C07319=1167.736,-18.694,-45.324,179.712,5.920,149.143
C07320=1167.731,-18.445,-45.336,179.714,5.921,149.143
C07321=1167.726,-18.196,-45.349,179.717,5.921,149.142
C07322=1167.720,-17.945,-45.362,179.719,5.922,149.141
C07323=1167.715,-17.695,-45.374,179.722,5.922,149.141
C07324=1167.710,-17.446,-45.387,179.724,5.923,149.140
C07325=1167.705,-17.197,-45.399,179.726,5.923,149.140
C07326=1167.700,-16.947,-45.412,179.728,5.923,149.139
C07327=1167.694,-16.697,-45.426,179.731,5.924,149.138
C07328=1167.689,-16.448,-45.438,179.733,5.925,149.138
C07329=1167.684,-16.198,-45.451,179.736,5.925,149.137
C07330=1167.680,-15.948,-45.464,179.738,5.926,149.137
C07331=1167.674,-15.698,-45.476,179.741,5.926,149.136
C07332=1167.668,-15.449,-45.489,179.743,5.927,149.135
C07333=1167.663,-15.200,-45.501,179.746,5.928,149.135
C07334=1167.659,-14.950,-45.514,179.748,5.928,149.134
C07335=1167.654,-14.700,-45.527,179.751,5.928,149.133
C07336=1167.648,-14.451,-45.540,179.753,5.929,149.133
C07337=1167.643,-14.201,-45.553,179.756,5.930,149.132
C07338=1167.638,-13.951,-45.566,179.758,5.930,149.132
C07339=1167.633,-13.702,-45.578,179.761,5.931,149.131
C07340=1167.627,-13.452,-45.592,179.763,5.931,149.130
C07341=1167.623,-13.202,-45.604,179.765,5.932,149.130
C07342=1167.617,-12.953,-45.617,179.768,5.933,149.129
C07343=1167.612,-12.703,-45.630,179.770,5.933,149.129
C07344=1167.607,-12.453,-45.643,179.773,5.934,149.128
C07345=1167.602,-12.204,-45.656,179.776,5.934,149.127
C07346=1167.596,-11.954,-45.669,179.778,5.935,149.127
C07347=1167.591,-11.704,-45.682,179.780,5.936,149.126
C07348=1167.587,-11.456,-45.695,179.783,5.936,149.126
C07349=1167.582,-11.206,-45.708,179.785,5.937,149.125
C07350=1167.576,-10.956,-45.722,179.788,5.937,149.124
C07351=1167.571,-10.707,-45.734,179.790,5.938,149.124
C07352=1167.566,-10.457,-45.747,179.793,5.939,149.123
C07353=1167.561,-10.207,-45.760,179.795,5.939,149.123
C07354=1167.556,-9.958,-45.773,179.798,5.940,149.122
C07355=1167.550,-9.707,-45.786,179.800,5.940,149.121
C07356=1167.545,-9.458,-45.799,179.802,5.941,149.121
C07357=1167.540,-9.209,-45.812,179.805,5.942,149.120
C07358=1167.535,-8.959,-45.826,179.807,5.942,149.120
C07359=1167.530,-8.710,-45.839,179.810,5.943,149.119
C07360=1167.525,-8.460,-45.851,179.813,5.943,149.118
C07361=1167.520,-8.210,-45.865,179.815,5.944,149.118
C07362=1167.515,-7.961,-45.877,179.817,5.945,149.117
C07363=1167.510,-7.711,-45.892,179.820,5.945,149.117
C07364=1167.504,-7.462,-45.904,179.822,5.946,149.116
C07365=1167.499,-7.212,-45.917,179.825,5.946,149.115
C07366=1167.494,-6.962,-45.930,179.827,5.947,149.115
C07367=1167.489,-6.713,-45.943,179.830,5.948,149.114
C07368=1167.484,-6.463,-45.957,179.832,5.948,149.114
C07369=1167.479,-6.214,-45.970,179.834,5.949,149.113
C07370=1167.474,-5.963,-45.983,179.837,5.949,149.112
C07371=1167.469,-5.714,-45.996,179.839,5.950,149.112
C07372=1167.463,-5.465,-46.010,179.842,5.951,149.111
C07373=1167.458,-5.215,-46.023,179.844,5.951,149.111
C07374=1167.453,-4.966,-46.035,179.847,5.952,149.110
C07375=1167.448,-4.716,-46.050,179.849,5.952,149.109
C07376=1167.443,-4.467,-46.062,179.852,5.953,149.109
C07377=1167.438,-4.216,-46.076,179.854,5.954,149.108
C07378=1167.433,-3.967,-46.088,179.856,5.954,149.108
C07379=1167.427,-3.718,-46.102,179.859,5.955,149.107
C07380=1167.423,-3.468,-46.115,179.862,5.955,149.106
C07381=1167.417,-3.218,-46.129,179.864,5.956,149.106
C07382=1167.413,-2.969,-46.142,179.867,5.957,149.105
C07383=1167.407,-2.719,-46.155,179.869,5.957,149.105
C07384=1167.402,-2.470,-46.170,179.871,5.958,149.104
C07385=1167.397,-2.220,-46.182,179.874,5.960,149.104
C07386=1167.391,-1.970,-46.196,179.877,5.960,149.103
C07387=1167.387,-1.721,-46.209,179.880,5.960,149.102
C07388=1167.381,-1.471,-46.223,179.882,5.961,149.102
C07389=1167.376,-1.222,-46.235,179.884,5.962,149.101
C07390=1167.371,-0.972,-46.250,179.887,5.963,149.101
C07391=1167.366,-0.723,-46.262,179.889,5.963,149.100
C07392=1167.361,-0.473,-46.276,179.892,5.963,149.099
C07393=1167.355,-0.223,-46.290,179.894,5.964,149.099
C07394=1167.351,0.026,-46.303,179.897,5.965,149.098
C07395=1167.345,0.276,-46.317,179.899,5.966,149.098
C07396=1167.341,0.525,-46.330,179.901,5.966,149.097
C07397=1167.335,0.775,-46.343,179.904,5.967,149.096
C07398=1167.330,1.024,-46.358,179.906,5.967,149.096
C07399=1167.325,1.274,-46.370,179.909,5.968,149.095
C07400=1167.320,1.523,-46.385,179.911,5.969,149.095
C07401=1167.314,1.794,-46.399,179.914,5.970,149.094
C07402=1167.309,2.062,-46.413,179.917,5.970,149.093
C07403=1167.304,2.331,-46.428,179.920,5.971,149.093
C07404=1167.298,2.601,-46.443,179.922,5.971,149.092
C07405=1167.292,2.850,-46.456,179.925,5.972,149.091
C07406=1167.288,3.100,-46.470,179.927,5.973,149.091
C07407=1167.283,3.350,-46.483,179.929,5.973,149.090
C07408=1167.277,3.599,-46.497,179.933,5.975,149.090
C07409=1167.273,3.849,-46.510,179.935,5.975,149.089
C07410=1167.267,4.098,-46.524,179.937,5.976,149.088
C07411=1167.262,4.348,-46.538,179.940,5.976,149.088
C07412=1167.257,4.597,-46.552,179.942,5.977,149.087
C07413=1167.252,4.847,-46.565,179.945,5.978,149.087
C07414=1167.247,5.097,-46.579,179.948,5.978,149.086
C07415=1167.241,5.346,-46.593,179.950,5.979,149.085
C07416=1167.237,5.596,-46.606,179.952,5.979,149.085
C07417=1167.232,5.846,-46.620,179.955,5.980,149.084
C07418=1167.226,6.095,-46.634,179.957,5.981,149.084
C07419=1167.221,6.345,-46.648,179.960,5.981,149.083
C07420=1167.216,6.594,-46.661,179.963,5.983,149.082
C07421=1167.211,6.844,-46.675,179.965,5.983,149.082
C07422=1167.206,7.093,-46.689,179.967,5.984,149.081
C07423=1167.201,7.343,-46.703,179.970,5.985,149.081
C07424=1167.196,7.592,-46.716,179.972,5.985,149.080
C07425=1167.191,7.842,-46.730,179.975,5.986,149.079
C07426=1167.186,8.091,-46.744,179.978,5.986,149.079
C07427=1167.181,8.341,-46.758,179.980,5.987,149.078
C07428=1167.176,8.590,-46.771,179.982,5.988,149.078
C07429=1167.171,8.840,-46.786,179.985,5.988,149.077
C07430=1167.166,9.090,-46.800,179.988,5.990,149.076
C07431=1167.160,9.339,-46.813,179.990,5.990,149.076
C07432=1167.155,9.589,-46.827,179.993,5.991,149.075
C07433=1167.150,9.839,-46.842,179.995,5.992,149.075
C07434=1167.145,10.087,-46.855,179.997,5.992,149.074
C07435=1167.140,10.338,-46.868,-180.000,5.993,149.073
C07436=1167.135,10.587,-46.883,-179.997,5.993,149.073
C07437=1167.130,10.836,-46.897,-179.995,5.994,149.072
C07438=1167.125,11.086,-46.911,-179.992,5.995,149.072
C07439=1167.120,11.336,-46.925,-179.990,5.996,149.071
C07440=1167.115,11.585,-46.939,-179.987,5.997,149.071
C07441=1167.110,11.835,-46.952,-179.985,5.998,149.070
C07442=1167.105,12.085,-46.966,-179.982,5.998,149.069
C07443=1167.100,12.334,-46.981,-179.980,5.998,149.069
C07444=1167.094,12.583,-46.995,-179.977,5.999,149.068
C07445=1167.089,12.833,-47.009,-179.975,6.000,149.068
C07446=1167.084,13.083,-47.023,-179.973,6.001,149.067
C07447=1167.079,13.332,-47.037,-179.969,6.002,149.066
C07448=1167.074,13.581,-47.051,-179.967,6.002,149.066
C07449=1167.068,13.832,-47.065,-179.965,6.003,149.065
C07450=1167.064,14.081,-47.079,-179.962,6.004,149.065
C07451=1167.059,14.331,-47.093,-179.960,6.004,149.064
C07452=1167.054,14.580,-47.107,-179.957,6.005,149.063
C07453=1167.049,14.830,-47.121,-179.955,6.006,149.063
C07454=1167.044,15.079,-47.135,-179.952,6.006,149.062
C07455=1167.039,15.329,-47.150,-179.949,6.008,149.062
C07456=1167.033,15.578,-47.163,-179.947,6.008,149.061
C07457=1167.028,15.828,-47.178,-179.944,6.009,149.060
C07458=1167.023,16.077,-47.192,-179.942,6.010,149.060
C07459=1167.018,16.327,-47.206,-179.939,6.010,149.059
C07460=1167.013,16.576,-47.220,-179.937,6.011,149.059
C07461=1167.008,16.826,-47.234,-179.935,6.011,149.058
C07462=1167.003,17.076,-47.249,-179.931,6.013,149.058
C07463=1166.998,17.325,-47.263,-179.929,6.014,149.057
C07464=1166.993,17.575,-47.277,-179.927,6.014,149.056
C07465=1166.987,17.824,-47.291,-179.924,6.015,149.056
C07466=1166.982,18.074,-47.306,-179.922,6.015,149.055
C07467=1166.978,18.323,-47.320,-179.919,6.016,149.055
C07468=1166.973,18.573,-47.335,-179.916,6.017,149.054
C07469=1166.968,18.822,-47.349,-179.914,6.018,149.053
C07470=1166.962,19.071,-47.363,-179.911,6.019,149.053
C07471=1166.957,19.321,-47.377,-179.909,6.019,149.052
C07472=1166.952,19.571,-47.392,-179.907,6.020,149.052
C07473=1166.948,19.820,-47.406,-179.904,6.021,149.051
C07474=1166.942,20.070,-47.421,-179.901,6.022,149.050
C07475=1166.937,20.320,-47.435,-179.899,6.023,149.050
C07476=1166.931,20.569,-47.449,-179.896,6.023,149.049
C07477=1166.927,20.818,-47.464,-179.894,6.024,149.049
C07478=1166.922,21.068,-47.478,-179.891,6.024,149.048
C07479=1166.917,21.318,-47.492,-179.889,6.025,149.048
C07480=1166.912,21.567,-47.507,-179.886,6.027,149.047
C07481=1166.907,21.817,-47.521,-179.883,6.027,149.046
C07482=1166.902,22.066,-47.536,-179.881,6.028,149.046
C07483=1166.897,22.315,-47.550,-179.878,6.028,149.045
C07484=1166.891,22.565,-47.565,-179.876,6.029,149.045
C07485=1166.886,22.815,-47.579,-179.873,6.031,149.044
C07486=1166.881,23.065,-47.593,-179.871,6.031,149.044
C07487=1166.876,23.314,-47.608,-179.868,6.032,149.043
C07488=1166.871,23.563,-47.623,-179.865,6.032,149.042
C07489=1166.866,23.813,-47.637,-179.863,6.033,149.042
C07490=1166.861,24.062,-47.652,-179.861,6.034,149.041
C07491=1166.856,24.312,-47.667,-179.858,6.035,149.041
C07492=1166.851,24.561,-47.681,-179.855,6.036,149.040
C07493=1166.846,24.811,-47.695,-179.853,6.037,149.040
C07494=1166.841,25.060,-47.710,-179.850,6.037,149.039
C07495=1166.836,25.310,-47.724,-179.848,6.038,149.038
C07496=1166.830,25.560,-47.739,-179.845,6.039,149.038
C07497=1166.826,25.809,-47.754,-179.842,6.040,149.037
C07498=1166.821,26.059,-47.768,-179.840,6.041,149.037
C07499=1166.816,26.308,-47.783,-179.838,6.041,149.036
C07500=1166.810,26.558,-47.798,-179.835,6.043,149.036
C07501=1166.805,26.807,-47.812,-179.832,6.043,149.035
C07502=1166.800,27.057,-47.827,-179.830,6.044,149.034
C07503=1166.796,27.306,-47.842,-179.827,6.044,149.034
C07504=1166.790,27.556,-47.857,-179.825,6.045,149.033
C07505=1166.785,27.825,-47.872,-179.822,6.047,149.033
C07506=1166.780,28.094,-47.888,-179.819,6.047,149.032
C07507=1166.774,28.363,-47.904,-179.816,6.048,149.031
C07508=1166.768,28.631,-47.920,-179.813,6.049,149.031
C07509=1166.764,28.880,-47.935,-179.811,6.050,149.030
C07510=1166.758,29.130,-47.950,-179.809,6.050,149.029
C07511=1166.753,29.380,-47.964,-179.806,6.052,149.029
C07512=1166.748,29.629,-47.979,-179.803,6.052,149.028
C07513=1166.743,29.879,-47.994,-179.801,6.053,149.028
C07514=1166.738,30.128,-48.009,-179.798,6.054,149.027
C07515=1166.733,30.378,-48.023,-179.796,6.055,149.027
C07516=1166.728,30.627,-48.039,-179.793,6.056,149.026
C07517=1166.723,30.877,-48.053,-179.790,6.056,149.025
C07518=1166.718,31.126,-48.068,-179.788,6.057,149.025
C07519=1166.713,31.375,-48.083,-179.786,6.058,149.024
C07520=1166.708,31.626,-48.098,-179.783,6.059,149.024
C07521=1166.704,31.875,-48.113,-179.780,6.060,149.023
C07522=1166.698,32.125,-48.128,-179.778,6.061,149.023
C07523=1166.693,32.374,-48.143,-179.775,6.061,149.022
C07524=1166.688,32.624,-48.157,-179.773,6.063,149.022
C07525=1166.683,32.873,-48.173,-179.770,6.063,149.021
C07526=1166.678,33.123,-48.187,-179.767,6.064,149.020
C07527=1166.673,33.372,-48.203,-179.765,6.065,149.020
C07528=1166.668,33.621,-48.218,-179.762,6.066,149.019
C07529=1166.663,33.871,-48.232,-179.760,6.067,149.019
C07530=1166.658,34.120,-48.247,-179.757,6.067,149.018
C07531=1166.653,34.369,-48.262,-179.755,6.068,149.017
C07532=1166.647,34.619,-48.277,-179.752,6.069,149.017
C07533=1166.643,34.869,-48.292,-179.750,6.070,149.016
C07534=1166.637,35.118,-48.308,-179.747,6.071,149.016
C07535=1166.632,35.368,-48.322,-179.745,6.071,149.015
C07536=1166.627,35.617,-48.338,-179.741,6.073,149.015
C07537=1166.623,35.867,-48.353,-179.739,6.073,149.014
C07538=1166.617,36.117,-48.368,-179.737,6.074,149.013
C07539=1166.613,36.366,-48.383,-179.733,6.075,149.013
C07540=1166.607,36.615,-48.399,-179.731,6.076,149.012
C07541=1166.602,36.865,-48.413,-179.729,6.077,149.012
C07542=1166.597,37.115,-48.428,-179.726,6.078,149.011
C07543=1166.592,37.364,-48.443,-179.723,6.079,149.011
C07544=1166.587,37.613,-48.459,-179.721,6.080,149.010
C07545=1166.582,37.863,-48.473,-179.718,6.080,149.009
C07546=1166.577,38.113,-48.489,-179.716,6.081,149.009
C07547=1166.572,38.362,-48.504,-179.713,6.082,149.008
C07548=1166.567,38.611,-48.520,-179.711,6.083,149.008
C07549=1166.562,38.860,-48.535,-179.708,6.084,149.007
C07550=1166.557,39.110,-48.550,-179.706,6.085,149.007
C07551=1166.552,39.360,-48.565,-179.703,6.086,149.006
C07552=1166.547,39.609,-48.580,-179.700,6.086,149.005
C07553=1166.543,39.859,-48.596,-179.698,6.087,149.005
C07554=1166.537,40.108,-48.611,-179.695,6.088,149.004
C07555=1166.532,40.358,-48.627,-179.693,6.089,149.004
C07556=1166.527,40.607,-48.642,-179.690,6.090,149.003
C07557=1166.521,40.857,-48.657,-179.687,6.091,149.003
C07558=1166.517,41.106,-48.672,-179.685,6.092,149.002
C07559=1166.512,41.356,-48.688,-179.682,6.093,149.002
C07560=1166.507,41.605,-48.703,-179.679,6.094,149.001
C07561=1166.502,41.854,-48.718,-179.677,6.095,149.000
C07562=1166.497,42.104,-48.734,-179.674,6.095,149.000
C07563=1166.491,42.353,-48.749,-179.672,6.096,148.999
C07564=1166.487,42.603,-48.765,-179.669,6.098,148.999
C07565=1166.482,42.852,-48.780,-179.667,6.098,148.998
C07566=1166.477,43.101,-48.795,-179.664,6.099,148.998
C07567=1166.472,43.351,-48.811,-179.662,6.101,148.997
C07568=1166.467,43.601,-48.827,-179.659,6.101,148.996
C07569=1166.462,43.850,-48.842,-179.656,6.102,148.996
C07570=1166.457,44.099,-48.857,-179.653,6.103,148.995
C07571=1166.452,44.349,-48.873,-179.651,6.104,148.995
C07572=1166.447,44.599,-48.888,-179.649,6.105,148.994
C07573=1166.442,44.848,-48.904,-179.645,6.106,148.994
C07574=1166.437,45.097,-48.920,-179.643,6.107,148.993
C07575=1166.431,45.347,-48.935,-179.641,6.107,148.992
C07576=1166.427,45.597,-48.951,-179.638,6.109,148.992
C07577=1166.422,45.846,-48.966,-179.635,6.109,148.991
C07578=1166.416,46.095,-48.982,-179.633,6.110,148.991
C07579=1166.412,46.344,-48.997,-179.630,6.112,148.990
C07580=1166.407,46.595,-49.013,-179.628,6.112,148.990
C07581=1166.402,46.844,-49.028,-179.625,6.113,148.989
C07582=1166.396,47.093,-49.044,-179.622,6.115,148.989
C07583=1166.392,47.342,-49.059,-179.620,6.115,148.988
C07584=1166.387,47.593,-49.075,-179.618,6.116,148.987
C07585=1166.382,47.841,-49.091,-179.614,6.117,148.987
C07586=1166.376,48.091,-49.107,-179.612,6.118,148.986
C07587=1166.372,48.341,-49.123,-179.610,6.119,148.986
C07588=1166.367,48.590,-49.138,-179.607,6.120,148.985
C07589=1166.362,48.839,-49.153,-179.604,6.121,148.985
C07590=1166.357,49.089,-49.169,-179.602,6.122,148.984
C07591=1166.352,49.338,-49.185,-179.599,6.123,148.983
C07592=1166.346,49.588,-49.201,-179.597,6.124,148.983
C07593=1166.342,49.837,-49.216,-179.594,6.124,148.982
C07594=1166.337,50.087,-49.232,-179.591,6.126,148.982
C07595=1166.331,50.336,-49.248,-179.589,6.126,148.981
C07596=1166.327,50.586,-49.264,-179.586,6.127,148.981
C07597=1166.322,50.835,-49.280,-179.583,6.129,148.980
C07598=1166.316,51.085,-49.295,-179.581,6.130,148.980
C07599=1166.312,51.334,-49.311,-179.578,6.130,148.979
C07600=1166.307,51.583,-49.327,-179.576,6.132,148.979
C07601=1166.302,51.833,-49.343,-179.573,6.132,148.978
C07602=1166.297,52.083,-49.359,-179.570,6.134,148.978
C07603=1166.292,52.331,-49.375,-179.568,6.134,148.977
C07604=1166.287,52.582,-49.391,-179.566,6.135,148.976
C07605=1166.282,52.831,-49.406,-179.562,6.137,148.976
C07606=1166.277,53.080,-49.423,-179.560,6.137,148.975
C07607=1166.272,53.330,-49.439,-179.557,6.138,148.975
C07608=1166.267,53.579,-49.454,-179.555,6.140,148.974
C07609=1166.262,53.847,-49.471,-179.552,6.140,148.974
C07610=1166.257,54.117,-49.488,-179.549,6.141,148.973
C07611=1166.251,54.384,-49.506,-179.547,6.142,148.972
C07612=1166.246,54.653,-49.523,-179.544,6.144,148.972
C07613=1166.241,54.903,-49.539,-179.541,6.144,148.971
C07614=1166.236,55.152,-49.555,-179.538,6.146,148.971
C07615=1166.231,55.401,-49.571,-179.536,6.147,148.970
C07616=1166.226,55.651,-49.587,-179.533,6.148,148.970
C07617=1166.221,55.900,-49.603,-179.531,6.149,148.969
C07618=1166.216,56.150,-49.619,-179.528,6.149,148.968
C07619=1166.211,56.399,-49.635,-179.525,6.151,148.968
C07620=1166.206,56.649,-49.651,-179.523,6.151,148.967
C07621=1166.201,56.898,-49.667,-179.520,6.153,148.967
C07622=1166.196,57.147,-49.683,-179.517,6.154,148.966
C07623=1166.191,57.397,-49.700,-179.515,6.154,148.966
C07624=1166.186,57.646,-49.715,-179.512,6.156,148.965
C07625=1166.181,57.896,-49.732,-179.510,6.157,148.965
C07626=1166.175,58.145,-49.748,-179.506,6.158,148.964
C07627=1166.171,58.395,-49.765,-179.504,6.159,148.964
C07628=1166.165,58.644,-49.780,-179.502,6.159,148.963
C07629=1166.161,58.894,-49.797,-179.499,6.161,148.962
C07630=1166.155,59.143,-49.813,-179.496,6.161,148.962
C07631=1166.151,59.393,-49.829,-179.494,6.163,148.961
C07632=1166.146,59.642,-49.845,-179.491,6.164,148.961
C07633=1166.141,59.891,-49.862,-179.489,6.165,148.960
C07634=1166.136,60.140,-49.878,-179.486,6.166,148.960
C07635=1166.131,60.390,-49.894,-179.483,6.167,148.959
C07636=1166.126,60.639,-49.910,-179.480,6.168,148.959
C07637=1166.121,60.889,-49.926,-179.478,6.169,148.958
C07638=1166.115,61.138,-49.943,-179.475,6.171,148.958
C07639=1166.111,61.388,-49.960,-179.473,6.171,148.957
C07640=1166.106,61.637,-49.975,-179.470,6.172,148.957
C07641=1166.101,61.887,-49.992,-179.467,6.173,148.956
C07642=1166.097,62.136,-50.009,-179.465,6.174,148.955
C07643=1166.091,62.386,-50.024,-179.462,6.175,148.955
C07644=1166.087,62.635,-50.041,-179.460,6.176,148.954
C07645=1166.081,62.884,-50.058,-179.457,6.178,148.954
C07646=1166.076,63.134,-50.074,-179.454,6.179,148.953
C07647=1166.071,63.383,-50.090,-179.452,6.179,148.953
C07648=1166.067,63.633,-50.107,-179.449,6.181,148.952
C07649=1166.062,63.881,-50.123,-179.446,6.181,148.951
C07650=1166.057,64.131,-50.139,-179.444,6.183,148.951
C07651=1166.052,64.381,-50.156,-179.441,6.184,148.951
C07652=1166.046,64.630,-50.173,-179.438,6.185,148.950
C07653=1166.042,64.879,-50.189,-179.436,6.186,148.950
C07654=1166.037,65.129,-50.205,-179.433,6.187,148.949
C07655=1166.031,65.379,-50.222,-179.431,6.188,148.948
C07656=1166.027,65.628,-50.239,-179.428,6.189,148.948
C07657=1166.022,65.877,-50.255,-179.425,6.190,148.947
C07658=1166.017,66.126,-50.272,-179.423,6.191,148.947
C07659=1166.012,66.376,-50.287,-179.420,6.193,148.946
C07660=1166.007,66.626,-50.305,-179.417,6.193,148.946
C07661=1166.002,66.875,-50.321,-179.415,6.195,148.945
C07662=1165.997,67.124,-50.338,-179.412,6.196,148.945
C07663=1165.992,67.374,-50.355,-179.409,6.197,148.944
C07664=1165.987,67.623,-50.371,-179.407,6.198,148.944
C07665=1165.982,67.872,-50.388,-179.404,6.199,148.943
C07666=1165.978,68.121,-50.404,-179.402,6.200,148.943
C07667=1165.973,68.371,-50.422,-179.399,6.201,148.942
C07668=1165.967,68.621,-50.437,-179.396,6.202,148.941
C07669=1165.963,68.870,-50.454,-179.393,6.203,148.941
C07670=1165.958,69.120,-50.471,-179.391,6.204,148.940
C07671=1165.953,69.369,-50.488,-179.388,6.206,148.940
C07672=1165.948,69.618,-50.504,-179.386,6.207,148.939
C07673=1165.943,69.868,-50.521,-179.383,6.207,148.939
C07674=1165.938,70.117,-50.538,-179.380,6.209,148.938
C07675=1165.933,70.366,-50.554,-179.378,6.210,148.938
C07676=1165.928,70.616,-50.572,-179.375,6.211,148.937
C07677=1165.923,70.865,-50.588,-179.373,6.212,148.937
C07678=1165.918,71.115,-50.605,-179.370,6.214,148.936
C07679=1165.913,71.364,-50.622,-179.367,6.214,148.936
C07680=1165.909,71.614,-50.639,-179.365,6.216,148.935
C07681=1165.903,71.863,-50.655,-179.362,6.216,148.934
C07682=1165.898,72.112,-50.672,-179.359,6.218,148.934
C07683=1165.893,72.362,-50.689,-179.357,6.218,148.933
C07684=1165.888,72.611,-50.706,-179.354,6.220,148.933
C07685=1165.884,72.860,-50.722,-179.352,6.221,148.933
C07686=1165.879,73.109,-50.740,-179.349,6.222,148.932
C07687=1165.874,73.359,-50.757,-179.346,6.223,148.931
C07688=1165.869,73.608,-50.774,-179.343,6.225,148.931
C07689=1165.864,73.857,-50.791,-179.341,6.225,148.930
C07690=1165.859,74.107,-50.808,-179.338,6.227,148.930
C07691=1165.854,74.357,-50.825,-179.336,6.228,148.929
C07692=1165.849,74.606,-50.841,-179.333,6.229,148.929
C07693=1165.844,74.855,-50.858,-179.330,6.230,148.928
C07694=1165.839,75.105,-50.876,-179.328,6.231,148.928
C07695=1165.835,75.354,-50.893,-179.324,6.233,148.927
C07696=1165.829,75.603,-50.910,-179.322,6.234,148.927
C07697=1165.824,75.853,-50.926,-179.320,6.235,148.926
C07698=1165.819,76.102,-50.944,-179.317,6.236,148.926
C07699=1165.815,76.351,-50.961,-179.314,6.238,148.925
C07700=1165.810,76.601,-50.978,-179.312,6.238,148.925
C07701=1165.805,76.850,-50.995,-179.309,6.240,148.924
C07702=1165.799,77.100,-51.012,-179.306,6.240,148.923
C07703=1165.795,77.348,-51.029,-179.303,6.242,148.923
C07704=1165.790,77.598,-51.046,-179.301,6.243,148.923
C07705=1165.785,77.848,-51.064,-179.298,6.244,148.922
C07706=1165.780,78.098,-51.080,-179.296,6.245,148.921
C07707=1165.775,78.346,-51.098,-179.293,6.246,148.921
C07708=1165.770,78.596,-51.115,-179.291,6.247,148.920
C07709=1165.765,78.845,-51.132,-179.288,6.249,148.920
C07710=1165.761,79.094,-51.149,-179.285,6.249,148.919
C07711=1165.756,79.344,-51.167,-179.282,6.251,148.919
C07712=1165.751,79.594,-51.184,-179.279,6.253,148.918
C07713=1165.746,79.861,-51.202,-179.277,6.253,148.918
C07714=1165.740,80.130,-51.221,-179.274,6.255,148.917
C07715=1165.735,80.399,-51.240,-179.271,6.256,148.917
C07716=1165.729,80.667,-51.258,-179.268,6.258,148.916
C07717=1165.725,80.916,-51.275,-179.266,6.259,148.916
C07718=1165.719,81.166,-51.293,-179.263,6.260,148.915
C07719=1165.715,81.415,-51.311,-179.260,6.261,148.915
C07720=1165.710,81.664,-51.327,-179.258,6.263,148.914
C07721=1165.705,81.914,-51.345,-179.255,6.263,148.914
C07722=1165.700,82.163,-51.363,-179.252,6.265,148.913
C07723=1165.695,82.412,-51.379,-179.250,6.265,148.912
C07724=1165.690,82.661,-51.397,-179.247,6.267,148.912
C07725=1165.685,82.911,-51.414,-179.244,6.269,148.912
C07726=1165.681,83.160,-51.431,-179.242,6.269,148.911
C07727=1165.675,83.410,-51.449,-179.239,6.271,148.911
C07728=1165.670,83.659,-51.467,-179.237,6.272,148.910
C07729=1165.665,83.909,-51.484,-179.234,6.273,148.909
C07730=1165.661,84.157,-51.501,-179.231,6.274,148.909
C07731=1165.656,84.407,-51.519,-179.228,6.275,148.908
C07732=1165.651,84.656,-51.537,-179.225,6.277,148.908
C07733=1165.646,84.906,-51.554,-179.223,6.278,148.908
C07734=1165.641,85.155,-51.571,-179.220,6.279,148.907
C07735=1165.637,85.404,-51.589,-179.218,6.280,148.906
C07736=1165.631,85.654,-51.607,-179.215,6.282,148.906
C07737=1165.626,85.903,-51.624,-179.212,6.283,148.905
C07738=1165.622,86.153,-51.641,-179.210,6.284,148.905
C07739=1165.617,86.402,-51.659,-179.207,6.285,148.904
C07740=1165.612,86.651,-51.677,-179.205,6.286,148.904
C07741=1165.606,86.900,-51.694,-179.202,6.288,148.903
C07742=1165.601,87.149,-51.712,-179.199,6.289,148.903
C07743=1165.596,87.399,-51.730,-179.196,6.290,148.902
C07744=1165.592,87.648,-51.747,-179.194,6.292,148.902
C07745=1165.587,87.897,-51.765,-179.191,6.292,148.901
C07746=1165.582,88.146,-51.783,-179.188,6.294,148.901
C07747=1165.577,88.396,-51.800,-179.186,6.296,148.900
C07748=1165.572,88.645,-51.818,-179.183,6.296,148.900
C07749=1165.568,88.895,-51.836,-179.180,6.298,148.899
C07750=1165.563,89.145,-51.853,-179.178,6.299,148.899
C07751=1165.558,89.394,-51.871,-179.175,6.300,148.898
C07752=1165.553,89.643,-51.889,-179.172,6.302,148.898
C07753=1165.549,89.892,-51.907,-179.170,6.302,148.897
C07754=1165.543,90.142,-51.924,-179.167,6.304,148.897
C07755=1165.538,90.391,-51.942,-179.165,6.305,148.896
C07756=1165.533,90.640,-51.960,-179.162,6.306,148.896
C07757=1165.529,90.890,-51.978,-179.159,6.308,148.895
C07758=1165.524,91.139,-51.996,-179.157,6.309,148.895
C07759=1165.518,91.389,-52.013,-179.153,6.310,148.894
C07760=1165.514,91.638,-52.031,-179.151,6.312,148.894
C07761=1165.509,91.887,-52.049,-179.149,6.313,148.893
C07762=1165.504,92.136,-52.067,-179.145,6.314,148.893
C07763=1165.499,92.385,-52.085,-179.143,6.315,148.892
C07764=1165.495,92.634,-52.103,-179.141,6.317,148.892
C07765=1165.490,92.883,-52.121,-179.137,6.318,148.891
C07766=1165.485,93.134,-52.138,-179.135,6.319,148.891
C07767=1165.480,93.383,-52.156,-179.132,6.321,148.890
C07768=1165.475,93.632,-52.174,-179.129,6.322,148.890
C07769=1165.470,93.881,-52.192,-179.127,6.323,148.889
C07770=1165.465,94.130,-52.210,-179.124,6.325,148.889
C07771=1165.460,94.380,-52.229,-179.121,6.326,148.888
C07772=1165.455,94.629,-52.247,-179.119,6.327,148.888
C07773=1165.450,94.878,-52.265,-179.116,6.329,148.888
C07774=1165.445,95.127,-52.283,-179.113,6.330,148.887
C07775=1165.441,95.377,-52.301,-179.111,6.331,148.886
C07776=1165.436,95.627,-52.319,-179.108,6.333,148.886
C07777=1165.431,95.876,-52.337,-179.105,6.334,148.885
C07778=1165.426,96.125,-52.355,-179.103,6.335,148.885
C07779=1165.421,96.374,-52.373,-179.100,6.337,148.885
C07780=1165.416,96.623,-52.391,-179.097,6.338,148.884
C07781=1165.411,96.872,-52.409,-179.095,6.339,148.884
C07782=1165.407,97.122,-52.427,-179.092,6.340,148.883
C07783=1165.402,97.371,-52.445,-179.089,6.342,148.882
C07784=1165.397,97.621,-52.463,-179.087,6.343,148.882
C07785=1165.391,97.870,-52.482,-179.084,6.344,148.882
C07786=1165.387,98.119,-52.500,-179.081,6.346,148.881
C07787=1165.382,98.369,-52.518,-179.079,6.347,148.881
C07788=1165.377,98.618,-52.536,-179.076,6.348,148.880
C07789=1165.373,98.867,-52.555,-179.073,6.350,148.880
C07790=1165.368,99.116,-52.573,-179.071,6.351,148.879
C07791=1165.363,99.365,-52.591,-179.068,6.352,148.879
C07792=1165.358,99.615,-52.610,-179.065,6.354,148.878
C07793=1165.353,99.865,-52.628,-179.063,6.355,148.878
C07794=1165.348,100.114,-52.646,-179.060,6.356,148.877
C07795=1165.343,100.362,-52.664,-179.057,6.358,148.877
C07796=1165.339,100.611,-52.682,-179.055,6.358,148.876
C07797=1165.333,100.862,-52.701,-179.052,6.360,148.876
C07798=1165.329,101.111,-52.719,-179.049,6.362,148.875
C07799=1165.324,101.360,-52.737,-179.047,6.363,148.875
C07800=1165.319,101.609,-52.756,-179.044,6.364,148.874
C07801=1165.315,101.858,-52.774,-179.041,6.366,148.874
C07802=1165.309,102.108,-52.793,-179.038,6.368,148.873
C07803=1165.304,102.357,-52.811,-179.036,6.368,148.873
C07804=1165.300,102.606,-52.829,-179.033,6.370,148.872
C07805=1165.295,102.856,-52.848,-179.030,6.372,148.872
C07806=1165.290,103.105,-52.866,-179.028,6.372,148.872
C07807=1165.285,103.354,-52.884,-179.025,6.374,148.871
C07808=1165.281,103.603,-52.903,-179.022,6.375,148.871
C07809=1165.275,103.853,-52.922,-179.020,6.376,148.870
C07810=1165.270,104.102,-52.940,-179.017,6.378,148.869
C07811=1165.266,104.351,-52.959,-179.014,6.379,148.869
C07812=1165.261,104.601,-52.977,-179.011,6.381,148.869
C07813=1165.256,104.850,-52.996,-179.009,6.382,148.868
C07814=1165.251,105.099,-53.014,-179.006,6.383,148.868
C07815=1165.247,105.349,-53.033,-179.003,6.385,148.867
C07816=1165.241,105.597,-53.052,-179.001,6.387,148.867
C07817=1165.236,105.866,-53.071,-178.998,6.387,148.866
C07818=1165.231,106.135,-53.092,-178.995,6.389,148.866
C07819=1165.226,106.403,-53.112,-178.992,6.390,148.865
C07820=1165.220,106.671,-53.132,-178.989,6.392,148.865
C07821=1165.215,106.920,-53.150,-178.987,6.394,148.864
C07822=1165.211,107.170,-53.169,-178.983,6.395,148.864
C07823=1165.206,107.419,-53.187,-178.981,6.396,148.863
C07824=1165.201,107.668,-53.206,-178.979,6.398,148.863
C07825=1165.196,107.918,-53.225,-178.976,6.399,148.862
C07826=1165.192,108.166,-53.244,-178.973,6.401,148.862
C07827=1165.187,108.417,-53.263,-178.971,6.402,148.861
C07828=1165.182,108.665,-53.281,-178.968,6.403,148.861
C07829=1165.176,108.915,-53.300,-178.965,6.405,148.861
C07830=1165.172,109.164,-53.319,-178.962,6.407,148.860
C07831=1165.167,109.413,-53.337,-178.960,6.407,148.860
C07832=1165.163,109.663,-53.357,-178.957,6.409,148.859
C07833=1165.158,109.911,-53.375,-178.954,6.411,148.859
C07834=1165.152,110.161,-53.394,-178.951,6.412,148.858
C07835=1165.148,110.410,-53.413,-178.949,6.413,148.858
C07836=1165.143,110.659,-53.432,-178.946,6.415,148.857
C07837=1165.139,110.909,-53.451,-178.944,6.417,148.857
C07838=1165.133,111.157,-53.470,-178.940,6.418,148.856
C07839=1165.128,111.407,-53.488,-178.938,6.420,148.856
C07840=1165.124,111.656,-53.508,-178.936,6.421,148.855
C07841=1165.119,111.905,-53.526,-178.933,6.422,148.855
C07842=1165.114,112.155,-53.545,-178.930,6.424,148.855
C07843=1165.109,112.403,-53.564,-178.927,6.425,148.854
C07844=1165.105,112.653,-53.584,-178.925,6.426,148.854
C07845=1165.100,112.902,-53.602,-178.922,6.428,148.853
C07846=1165.095,113.152,-53.621,-178.919,6.430,148.853
C07847=1165.090,113.401,-53.640,-178.916,6.431,148.852
C07848=1165.085,113.650,-53.658,-178.914,6.432,148.852
C07849=1165.080,113.899,-53.678,-178.911,6.434,148.851
C07850=1165.075,114.148,-53.697,-178.909,6.435,148.851
C07851=1165.071,114.398,-53.716,-178.905,6.437,148.850
C07852=1165.065,114.646,-53.736,-178.903,6.438,148.850
C07853=1165.061,114.896,-53.754,-178.901,6.439,148.849
C07854=1165.056,115.145,-53.773,-178.898,6.441,148.849
C07855=1165.052,115.394,-53.792,-178.895,6.443,148.849
C07856=1165.046,115.643,-53.812,-178.892,6.444,148.848
C07857=1165.042,115.893,-53.831,-178.889,6.446,148.848
C07858=1165.037,116.142,-53.849,-178.887,6.447,148.847
C07859=1165.032,116.392,-53.869,-178.884,6.448,148.847
C07860=1165.027,116.640,-53.888,-178.881,6.450,148.846
C07861=1165.023,116.890,-53.907,-178.878,6.452,148.846
C07862=1165.017,117.139,-53.927,-178.876,6.453,148.845
C07863=1165.012,117.388,-53.946,-178.874,6.454,148.845
C07864=1165.008,117.637,-53.965,-178.871,6.456,148.845
C07865=1165.003,117.886,-53.985,-178.868,6.457,148.844
C07866=1164.998,118.136,-54.004,-178.865,6.459,148.844
C07867=1164.993,118.385,-54.022,-178.862,6.461,148.843
C07868=1164.989,118.635,-54.042,-178.860,6.462,148.843
C07869=1164.983,118.883,-54.061,-178.857,6.463,148.842
C07870=1164.979,119.133,-54.081,-178.854,6.465,148.842
C07871=1164.974,119.382,-54.100,-178.852,6.466,148.841
C07872=1164.969,119.631,-54.119,-178.849,6.468,148.841
C07873=1164.965,119.881,-54.139,-178.846,6.470,148.840
C07874=1164.959,120.130,-54.158,-178.844,6.471,148.840
C07875=1164.955,120.379,-54.177,-178.841,6.472,148.840
C07876=1164.950,120.628,-54.197,-178.838,6.474,148.839
C07877=1164.945,120.877,-54.216,-178.835,6.476,148.839
C07878=1164.940,121.127,-54.236,-178.833,6.477,148.838
C07879=1164.936,121.375,-54.255,-178.830,6.479,148.838
C07880=1164.931,121.625,-54.274,-178.828,6.480,148.837
C07881=1164.927,121.874,-54.295,-178.825,6.481,148.837
C07882=1164.921,122.123,-54.314,-178.822,6.483,148.836
C07883=1164.917,122.372,-54.334,-178.819,6.485,148.836
C07884=1164.911,122.621,-54.353,-178.816,6.486,148.836
C07885=1164.907,122.870,-54.372,-178.814,6.488,148.835
C07886=1164.902,123.120,-54.392,-178.812,6.489,148.835
C07887=1164.897,123.369,-54.411,-178.808,6.490,148.834
C07888=1164.892,123.618,-54.431,-178.806,6.492,148.834
C07889=1164.888,123.867,-54.451,-178.803,6.494,148.833
C07890=1164.883,124.116,-54.470,-178.800,6.496,148.833
C07891=1164.878,124.366,-54.490,-178.798,6.497,148.833
C07892=1164.874,124.615,-54.509,-178.795,6.499,148.832
C07893=1164.868,124.864,-54.528,-178.792,6.500,148.832
C07894=1164.864,125.113,-54.549,-178.790,6.501,148.831
C07895=1164.859,125.363,-54.568,-178.787,6.503,148.831
C07896=1164.855,125.612,-54.588,-178.784,6.505,148.830
C07897=1164.849,125.861,-54.607,-178.781,6.506,148.830
C07898=1164.845,126.110,-54.628,-178.779,6.508,148.830
C07899=1164.840,126.359,-54.647,-178.776,6.510,148.829
C07900=1164.835,126.608,-54.666,-178.773,6.511,148.829
C07901=1164.830,126.858,-54.686,-178.771,6.512,148.828
C07902=1164.825,127.107,-54.706,-178.768,6.514,148.828
C07903=1164.821,127.356,-54.726,-178.765,6.516,148.827
C07904=1164.815,127.605,-54.745,-178.763,6.517,148.827
C07905=1164.811,127.854,-54.766,-178.760,6.519,148.827
C07906=1164.807,128.103,-54.785,-178.757,6.520,148.826
C07907=1164.802,128.353,-54.805,-178.754,6.522,148.826
C07908=1164.797,128.601,-54.825,-178.751,6.524,148.825
C07909=1164.792,128.851,-54.845,-178.749,6.525,148.825
C07910=1164.787,129.100,-54.865,-178.746,6.527,148.824
C07911=1164.783,129.350,-54.885,-178.744,6.528,148.824
C07912=1164.777,129.599,-54.904,-178.741,6.530,148.824
C07913=1164.773,129.848,-54.924,-178.738,6.531,148.823
C07914=1164.768,130.097,-54.944,-178.735,6.533,148.823
C07915=1164.764,130.346,-54.965,-178.732,6.535,148.822
C07916=1164.758,130.595,-54.984,-178.730,6.537,148.822
C07917=1164.754,130.844,-55.004,-178.727,6.538,148.821
C07918=1164.749,131.093,-55.024,-178.724,6.540,148.821
C07919=1164.745,131.342,-55.044,-178.722,6.541,148.821
C07920=1164.740,131.592,-55.064,-178.719,6.543,148.820
C07921=1164.734,131.861,-55.086,-178.716,6.544,148.820
C07922=1164.730,132.129,-55.107,-178.713,6.547,148.819
C07923=1164.724,132.398,-55.129,-178.710,6.548,148.819
C07924=1164.719,132.667,-55.150,-178.707,6.550,148.818
C07925=1164.714,132.915,-55.170,-178.704,6.551,148.818
C07926=1164.710,133.164,-55.190,-178.702,6.553,148.817
C07927=1164.705,133.413,-55.210,-178.699,6.555,148.817
C07928=1164.700,133.663,-55.231,-178.696,6.557,148.817
C07929=1164.695,133.912,-55.251,-178.694,6.557,148.816
C07930=1164.690,134.161,-55.271,-178.691,6.559,148.816
C07931=1164.685,134.409,-55.291,-178.689,6.561,148.815
C07932=1164.681,134.659,-55.311,-178.686,6.563,148.815
C07933=1164.676,134.908,-55.331,-178.683,6.564,148.814
C07934=1164.671,135.158,-55.351,-178.680,6.566,148.814
C07935=1164.666,135.407,-55.372,-178.677,6.568,148.814
C07936=1164.662,135.656,-55.392,-178.675,6.569,148.813
C07937=1164.657,135.905,-55.412,-178.672,6.571,148.813
C07938=1164.652,136.154,-55.433,-178.669,6.573,148.812
C07939=1164.648,136.403,-55.453,-178.667,6.574,148.812
C07940=1164.642,136.652,-55.473,-178.664,6.576,148.812
C07941=1164.638,136.901,-55.493,-178.661,6.578,148.811
C07942=1164.633,137.150,-55.514,-178.659,6.580,148.811
C07943=1164.628,137.399,-55.534,-178.656,6.581,148.811
C07944=1164.624,137.648,-55.555,-178.653,6.583,148.810
C07945=1164.619,137.898,-55.574,-178.650,6.584,148.810
C07946=1164.614,138.147,-55.595,-178.648,6.585,148.809
C07947=1164.609,138.396,-55.616,-178.645,6.587,148.809
C07948=1164.605,138.645,-55.636,-178.642,6.589,148.808
C07949=1164.600,138.894,-55.657,-178.640,6.591,148.808
C07950=1164.595,139.144,-55.677,-178.637,6.592,148.808
C07951=1164.591,139.393,-55.697,-178.634,6.594,148.807
C07952=1164.585,139.642,-55.718,-178.632,6.596,148.807
C07953=1164.581,139.891,-55.738,-178.629,6.598,148.806
C07954=1164.577,140.140,-55.759,-178.626,6.599,148.806
C07955=1164.571,140.389,-55.780,-178.623,6.601,148.806
C07956=1164.567,140.638,-55.800,-178.621,6.603,148.805
C07957=1164.562,140.888,-55.820,-178.618,6.604,148.805
C07958=1164.557,141.137,-55.841,-178.615,6.606,148.804
C07959=1164.553,141.386,-55.861,-178.612,6.608,148.804
C07960=1164.548,141.635,-55.881,-178.609,6.609,148.803
C07961=1164.543,141.884,-55.902,-178.607,6.611,148.803
C07962=1164.538,142.133,-55.923,-178.604,6.613,148.803
C07963=1164.533,142.382,-55.944,-178.601,6.615,148.802
C07964=1164.529,142.631,-55.964,-178.599,6.616,148.802
C07965=1164.524,142.880,-55.984,-178.596,6.618,148.802
C07966=1164.519,143.130,-56.005,-178.593,6.620,148.801
C07967=1164.515,143.379,-56.026,-178.591,6.621,148.801
C07968=1164.510,143.628,-56.047,-178.588,6.623,148.800
C07969=1164.505,143.877,-56.067,-178.585,6.625,148.800
C07970=1164.500,144.126,-56.088,-178.582,6.627,148.800
C07971=1164.496,144.375,-56.108,-178.580,6.628,148.799
C07972=1164.490,144.624,-56.129,-178.577,6.630,148.799
C07973=1164.486,144.873,-56.150,-178.574,6.632,148.798
C07974=1164.481,145.122,-56.171,-178.572,6.634,148.798
C07975=1164.477,145.371,-56.192,-178.569,6.635,148.798
C07976=1164.472,145.620,-56.213,-178.566,6.637,148.797
C07977=1164.467,145.869,-56.233,-178.564,6.639,148.797
C07978=1164.462,146.118,-56.254,-178.561,6.641,148.797
C07979=1164.458,146.368,-56.275,-178.558,6.642,148.796
C07980=1164.453,146.617,-56.296,-178.555,6.644,148.796
C07981=1164.449,146.865,-56.317,-178.553,6.646,148.795
C07982=1164.444,147.115,-56.338,-178.550,6.648,148.795
C07983=1164.439,147.364,-56.358,-178.547,6.649,148.795
C07984=1164.434,147.613,-56.379,-178.545,6.651,148.794
C07985=1164.429,147.862,-56.400,-178.542,6.653,148.794
C07986=1164.425,148.111,-56.421,-178.539,6.654,148.793
C07987=1164.419,148.360,-56.442,-178.537,6.656,148.793
C07988=1164.416,148.609,-56.463,-178.534,6.658,148.793
C07989=1164.410,148.859,-56.484,-178.531,6.660,148.792
C07990=1164.406,149.107,-56.506,-178.528,6.661,148.792
C07991=1164.401,149.356,-56.526,-178.526,6.663,148.792
C07992=1164.396,149.606,-56.547,-178.523,6.665,148.791
C07993=1164.392,149.854,-56.567,-178.520,6.667,148.791
C07994=1164.387,150.103,-56.589,-178.518,6.668,148.790
C07995=1164.382,150.353,-56.610,-178.515,6.670,148.790
C07996=1164.378,150.602,-56.631,-178.512,6.673,148.790
C07997=1164.373,150.851,-56.652,-178.509,6.674,148.789
C07998=1164.368,151.100,-56.673,-178.506,6.676,148.789
C07999=1164.364,151.348,-56.694,-178.504,6.678,148.789
C08000=1164.359,151.598,-56.716,-178.501,6.680,148.788
C08001=1164.354,151.847,-56.737,-178.498,6.681,148.788
C08002=1164.349,152.096,-56.758,-178.495,6.683,148.787
C08003=1164.344,152.345,-56.779,-178.493,6.685,148.787
C08004=1164.340,152.594,-56.800,-178.490,6.687,148.787
C08005=1164.335,152.844,-56.822,-178.487,6.688,148.786
C08006=1164.330,153.093,-56.843,-178.485,6.690,148.786
C08007=1164.326,153.341,-56.864,-178.482,6.692,148.786
C08008=1164.321,153.591,-56.885,-178.479,6.694,148.785
C08009=1164.316,153.839,-56.906,-178.477,6.695,148.785
C08010=1164.311,154.089,-56.928,-178.474,6.697,148.784
C08011=1164.307,154.337,-56.949,-178.471,6.699,148.784
C08012=1164.302,154.587,-56.970,-178.469,6.701,148.784
C08013=1164.297,154.835,-56.992,-178.465,6.703,148.783
C08014=1164.292,155.085,-57.013,-178.463,6.705,148.783
C08015=1164.287,155.334,-57.035,-178.460,6.707,148.782
C08016=1164.283,155.582,-57.056,-178.457,6.708,148.782
C08017=1164.278,155.832,-57.077,-178.454,6.710,148.782
C08018=1164.274,156.081,-57.099,-178.452,6.712,148.781
C08019=1164.269,156.330,-57.120,-178.449,6.714,148.781
C08020=1164.264,156.579,-57.141,-178.446,6.715,148.781
C08021=1164.260,156.828,-57.163,-178.444,6.717,148.780
C08022=1164.255,157.077,-57.184,-178.441,6.719,148.780
C08023=1164.250,157.326,-57.205,-178.438,6.721,148.779
C08024=1164.245,157.575,-57.226,-178.435,6.723,148.779
C08025=1164.240,157.844,-57.250,-178.432,6.725,148.779
C08026=1164.235,158.113,-57.273,-178.430,6.727,148.778
C08027=1164.230,158.382,-57.297,-178.426,6.729,148.778
C08028=1164.225,158.651,-57.320,-178.424,6.731,148.778
C08029=1164.221,158.901,-57.341,-178.421,6.733,148.777
C08030=1164.216,159.149,-57.363,-178.418,6.734,148.777
C08031=1164.211,159.398,-57.385,-178.416,6.736,148.777
C08032=1164.206,159.648,-57.406,-178.413,6.738,148.776
C08033=1164.201,159.896,-57.428,-178.410,6.740,148.776
C08034=1164.197,160.145,-57.449,-178.407,6.743,148.776
C08035=1164.192,160.394,-57.472,-178.405,6.744,148.775
C08036=1164.187,160.643,-57.493,-178.402,6.746,148.775
C08037=1164.182,160.892,-57.514,-178.399,6.748,148.775
C08038=1164.178,161.142,-57.536,-178.397,6.750,148.774
C08039=1164.173,161.390,-57.558,-178.394,6.751,148.774
C08040=1164.169,161.640,-57.580,-178.391,6.753,148.773
C08041=1164.164,161.888,-57.602,-178.389,6.755,148.773
C08042=1164.159,162.137,-57.623,-178.385,6.757,148.773
C08043=1164.155,162.387,-57.645,-178.383,6.759,148.772
C08044=1164.150,162.635,-57.666,-178.380,6.761,148.772
C08045=1164.145,162.885,-57.688,-178.377,6.763,148.772
C08046=1164.141,163.133,-57.710,-178.375,6.765,148.771
C08047=1164.136,163.382,-57.732,-178.372,6.766,148.771
C08048=1164.131,163.631,-57.754,-178.370,6.768,148.771
C08049=1164.127,163.880,-57.775,-178.367,6.770,148.770
C08050=1164.122,164.129,-57.798,-178.364,6.772,148.770
C08051=1164.117,164.378,-57.819,-178.361,6.774,148.770
C08052=1164.113,164.627,-57.841,-178.358,6.776,148.769
C08053=1164.108,164.876,-57.863,-178.356,6.778,148.769
C08054=1164.104,165.125,-57.885,-178.353,6.779,148.768
C08055=1164.099,165.374,-57.907,-178.351,6.782,148.768
C08056=1164.094,165.623,-57.929,-178.347,6.784,148.768
C08057=1164.089,165.872,-57.951,-178.345,6.786,148.768
C08058=1164.084,166.121,-57.973,-178.342,6.788,148.767
C08059=1164.080,166.370,-57.995,-178.339,6.789,148.767
C08060=1164.075,166.619,-58.016,-178.337,6.791,148.766
C08061=1164.071,166.868,-58.038,-178.334,6.793,148.766
C08062=1164.066,167.117,-58.060,-178.331,6.795,148.766
C08063=1164.061,167.367,-58.083,-178.328,6.797,148.765
C08064=1164.056,167.615,-58.104,-178.326,6.799,148.765
C08065=1164.052,167.864,-58.127,-178.323,6.801,148.765
C08066=1164.047,168.113,-58.149,-178.320,6.803,148.764
C08067=1164.043,168.362,-58.171,-178.318,6.805,148.764
C08068=1164.038,168.611,-58.193,-178.314,6.807,148.764
C08069=1164.033,168.860,-58.215,-178.312,6.809,148.763
C08070=1164.028,169.109,-58.237,-178.309,6.811,148.763
C08071=1164.024,169.358,-58.260,-178.307,6.813,148.763
C08072=1164.019,169.607,-58.282,-178.304,6.814,148.762
C08073=1164.015,169.856,-58.304,-178.301,6.816,148.762
C08074=1164.010,170.105,-58.326,-178.298,6.819,148.762
C08075=1164.005,170.354,-58.348,-178.295,6.821,148.761
C08076=1164.001,170.603,-58.371,-178.293,6.822,148.761
C08077=1163.996,170.852,-58.393,-178.290,6.824,148.761
C08078=1163.992,171.101,-58.415,-178.288,6.826,148.761
C08079=1163.986,171.350,-58.437,-178.285,6.829,148.760
C08080=1163.982,171.599,-58.460,-178.282,6.830,148.760
C08081=1163.978,171.848,-58.482,-178.279,6.832,148.759
C08082=1163.972,172.097,-58.504,-178.277,6.834,148.759
C08083=1163.968,172.346,-58.527,-178.274,6.836,148.759
C08084=1163.963,172.594,-58.549,-178.271,6.839,148.759
C08085=1163.958,172.844,-58.571,-178.268,6.840,148.758
C08086=1163.954,173.093,-58.594,-178.266,6.842,148.758
C08087=1163.950,173.341,-58.616,-178.263,6.844,148.757
C08088=1163.945,173.590,-58.639,-178.260,6.846,148.757
C08089=1163.940,173.839,-58.661,-178.257,6.849,148.757
C08090=1163.936,174.088,-58.683,-178.255,6.850,148.757
C08091=1163.931,174.337,-58.706,-178.252,6.852,148.756
C08092=1163.926,174.586,-58.728,-178.249,6.854,148.756
C08093=1163.921,174.835,-58.751,-178.246,6.856,148.756
C08094=1163.917,175.084,-58.773,-178.243,6.858,148.755
C08095=1163.912,175.333,-58.796,-178.241,6.860,148.755
C08096=1163.908,175.582,-58.818,-178.239,6.862,148.755
C08097=1163.904,175.831,-58.841,-178.236,6.864,148.754
C08098=1163.898,176.080,-58.863,-178.233,6.866,148.754
C08099=1163.894,176.328,-58.886,-178.230,6.868,148.754
C08100=1163.889,176.578,-58.909,-178.228,6.870,148.753
C08101=1163.884,176.826,-58.931,-178.225,6.872,148.753
C08102=1163.879,177.076,-58.954,-178.222,6.875,148.753
C08103=1163.875,177.324,-58.977,-178.219,6.876,148.752
C08104=1163.870,177.574,-58.999,-178.216,6.878,148.752
C08105=1163.866,177.822,-59.022,-178.214,6.880,148.752
C08106=1163.861,178.071,-59.045,-178.211,6.883,148.752
C08107=1163.857,178.320,-59.067,-178.208,6.885,148.751
C08108=1163.852,178.569,-59.090,-178.206,6.886,148.751
C08109=1163.847,178.818,-59.112,-178.203,6.888,148.750
C08110=1163.843,179.067,-59.135,-178.200,6.891,148.750
C08111=1163.839,179.316,-59.158,-178.197,6.893,148.750
C08112=1163.833,179.565,-59.180,-178.195,6.894,148.750
C08113=1163.829,179.814,-59.203,-178.192,6.896,148.749
C08114=1163.824,180.063,-59.227,-178.189,6.899,148.749
C08115=1163.820,180.312,-59.250,-178.187,6.901,148.749
C08116=1163.815,180.560,-59.272,-178.184,6.903,148.748
C08117=1163.810,180.809,-59.295,-178.181,6.904,148.748
C08118=1163.806,181.058,-59.318,-178.178,6.907,148.748
C08119=1163.801,181.308,-59.340,-178.176,6.909,148.748
C08120=1163.796,181.556,-59.363,-178.173,6.911,148.747
C08121=1163.792,181.805,-59.386,-178.170,6.913,148.747
C08122=1163.787,182.054,-59.410,-178.168,6.916,148.747
C08123=1163.783,182.303,-59.433,-178.165,6.917,148.746
C08124=1163.778,182.552,-59.455,-178.162,6.919,148.746
C08125=1163.773,182.800,-59.478,-178.159,6.922,148.746
C08126=1163.769,183.049,-59.501,-178.156,6.923,148.745
C08127=1163.764,183.298,-59.524,-178.154,6.925,148.745
C08128=1163.760,183.547,-59.547,-178.151,6.927,148.745
C08129=1163.754,183.817,-59.572,-178.148,6.930,148.744
C08130=1163.750,184.086,-59.597,-178.145,6.932,148.744
C08131=1163.744,184.356,-59.622,-178.142,6.934,148.744
C08132=1163.739,184.626,-59.647,-178.139,6.937,148.743
C08133=1163.735,184.875,-59.670,-178.137,6.939,148.743
C08134=1163.730,185.124,-59.693,-178.134,6.941,148.743
C08135=1163.726,185.373,-59.716,-178.131,6.943,148.743
C08136=1163.722,185.621,-59.739,-178.129,6.945,148.742
C08137=1163.716,185.870,-59.762,-178.126,6.947,148.742
C08138=1163.712,186.119,-59.786,-178.123,6.949,148.742
C08139=1163.707,186.368,-59.809,-178.120,6.951,148.741
C08140=1163.702,186.617,-59.832,-178.118,6.954,148.741
C08141=1163.698,186.866,-59.855,-178.115,6.955,148.741
C08142=1163.694,187.115,-59.878,-178.112,6.958,148.741
C08143=1163.689,187.364,-59.902,-178.110,6.960,148.740
C08144=1163.684,187.613,-59.925,-178.107,6.962,148.740
C08145=1163.680,187.862,-59.948,-178.104,6.964,148.740
C08146=1163.675,188.110,-59.971,-178.101,6.966,148.739
C08147=1163.670,188.359,-59.994,-178.099,6.968,148.739
C08148=1163.666,188.608,-60.018,-178.095,6.971,148.739
C08149=1163.661,188.856,-60.042,-178.093,6.973,148.739
C08150=1163.657,189.105,-60.065,-178.091,6.975,148.738
C08151=1163.652,189.354,-60.088,-178.087,6.977,148.738
C08152=1163.647,189.603,-60.112,-178.085,6.979,148.738
C08153=1163.642,189.852,-60.135,-178.082,6.981,148.737
C08154=1163.638,190.101,-60.158,-178.079,6.984,148.737
C08155=1163.634,190.350,-60.181,-178.076,6.985,148.737
C08156=1163.629,190.599,-60.205,-178.074,6.987,148.737
C08157=1163.625,190.848,-60.229,-178.071,6.990,148.737
C08158=1163.620,191.097,-60.252,-178.068,6.992,148.736
C08159=1163.615,191.346,-60.275,-178.066,6.994,148.736
C08160=1163.611,191.594,-60.299,-178.063,6.997,148.736
C08161=1163.606,191.843,-60.323,-178.060,6.998,148.735
C08162=1163.602,192.092,-60.346,-178.058,7.000,148.735
C08163=1163.597,192.341,-60.370,-178.055,7.003,148.735
C08164=1163.592,192.590,-60.394,-178.052,7.005,148.735
C08165=1163.588,192.839,-60.417,-178.049,7.007,148.734
C08166=1163.583,193.088,-60.440,-178.047,7.009,148.734
C08167=1163.579,193.336,-60.464,-178.044,7.011,148.734
C08168=1163.574,193.585,-60.488,-178.041,7.013,148.733
C08169=1163.569,193.834,-60.511,-178.038,7.016,148.733
C08170=1163.565,194.082,-60.535,-178.036,7.018,148.733
C08171=1163.560,194.332,-60.559,-178.033,7.020,148.733
C08172=1163.555,194.581,-60.582,-178.030,7.022,148.732
C08173=1163.551,194.829,-60.606,-178.028,7.024,148.732
C08174=1163.546,195.078,-60.629,-178.024,7.027,148.732
C08175=1163.542,195.326,-60.653,-178.022,7.029,148.732
C08176=1163.537,195.575,-60.677,-178.019,7.031,148.731
C08177=1163.533,195.824,-60.700,-178.016,7.033,148.731
C08178=1163.528,196.073,-60.724,-178.014,7.035,148.731
C08179=1163.523,196.322,-60.748,-178.011,7.038,148.730
C08180=1163.518,196.571,-60.772,-178.009,7.040,148.730
C08181=1163.514,196.820,-60.796,-178.006,7.042,148.730
C08182=1163.510,197.069,-60.820,-178.003,7.044,148.730
C08183=1163.505,197.318,-60.843,-178.000,7.047,148.730
C08184=1163.501,197.566,-60.867,-177.998,7.048,148.729
C08185=1163.496,197.815,-60.891,-177.994,7.051,148.729
C08186=1163.492,198.064,-60.915,-177.992,7.053,148.729
C08187=1163.487,198.312,-60.939,-177.989,7.056,148.728
C08188=1163.482,198.561,-60.963,-177.987,7.058,148.728
C08189=1163.477,198.810,-60.987,-177.984,7.059,148.728
C08190=1163.473,199.059,-61.010,-177.981,7.062,148.728
C08191=1163.469,199.308,-61.035,-177.979,7.064,148.727
C08192=1163.465,199.556,-61.059,-177.975,7.067,148.727
C08193=1163.459,199.806,-61.083,-177.973,7.068,148.727
C08194=1163.455,200.054,-61.107,-177.971,7.071,148.727
C08195=1163.450,200.303,-61.131,-177.967,7.073,148.726
C08196=1163.446,200.552,-61.154,-177.965,7.075,148.726
C08197=1163.442,200.801,-61.179,-177.962,7.078,148.726
C08198=1163.437,201.049,-61.203,-177.959,7.080,148.726
C08199=1163.432,201.298,-61.227,-177.957,7.082,148.725
C08200=1163.428,201.547,-61.251,-177.954,7.084,148.725
C08201=1163.423,201.795,-61.275,-177.952,7.086,148.725
C08202=1163.419,202.045,-61.300,-177.948,7.089,148.725
C08203=1163.414,202.294,-61.323,-177.946,7.091,148.725
C08204=1163.410,202.542,-61.347,-177.943,7.094,148.724
C08205=1163.404,202.791,-61.372,-177.940,7.096,148.724
C08206=1163.400,203.039,-61.396,-177.938,7.098,148.724
C08207=1163.396,203.289,-61.420,-177.935,7.100,148.723
C08208=1163.391,203.538,-61.445,-177.932,7.102,148.723
C08209=1163.386,203.786,-61.469,-177.929,7.105,148.723
C08210=1163.382,204.035,-61.493,-177.927,7.107,148.723
C08211=1163.377,204.284,-61.518,-177.924,7.110,148.723
C08212=1163.373,204.532,-61.542,-177.921,7.111,148.722
C08213=1163.369,204.781,-61.566,-177.919,7.114,148.722
C08214=1163.363,205.030,-61.590,-177.916,7.116,148.722
C08215=1163.359,205.279,-61.614,-177.913,7.118,148.722
C08216=1163.355,205.528,-61.638,-177.910,7.121,148.721
C08217=1163.350,205.776,-61.663,-177.908,7.123,148.721
C08218=1163.346,206.025,-61.687,-177.905,7.126,148.721
C08219=1163.341,206.274,-61.712,-177.902,7.127,148.720
C08220=1163.337,206.523,-61.736,-177.899,7.130,148.720
C08221=1163.331,206.771,-61.761,-177.897,7.132,148.720
C08222=1163.327,207.020,-61.785,-177.894,7.135,148.720
C08223=1163.323,207.269,-61.809,-177.891,7.137,148.720
C08224=1163.318,207.518,-61.834,-177.889,7.139,148.719
C08225=1163.314,207.766,-61.858,-177.886,7.141,148.719
C08226=1163.309,208.016,-61.883,-177.884,7.144,148.719
C08227=1163.305,208.264,-61.907,-177.880,7.146,148.719
C08228=1163.300,208.513,-61.932,-177.878,7.148,148.719
C08229=1163.296,208.762,-61.956,-177.875,7.151,148.718
C08230=1163.291,209.010,-61.981,-177.872,7.153,148.718
C08231=1163.286,209.259,-62.005,-177.869,7.156,148.718
C08232=1163.282,209.508,-62.031,-177.867,7.157,148.717
C08233=1163.277,209.778,-62.057,-177.864,7.160,148.717
C08234=1163.272,210.049,-62.084,-177.861,7.163,148.717
C08235=1163.267,210.320,-62.111,-177.857,7.165,148.717
C08236=1163.262,210.590,-62.137,-177.855,7.168,148.717
C08237=1163.258,210.839,-62.162,-177.852,7.170,148.716
C08238=1163.253,211.087,-62.187,-177.850,7.172,148.716
C08239=1163.248,211.336,-62.212,-177.847,7.175,148.716
C08240=1163.244,211.585,-62.236,-177.844,7.177,148.716
C08241=1163.239,211.833,-62.261,-177.841,7.180,148.715
C08242=1163.235,212.083,-62.285,-177.839,7.182,148.715
C08243=1163.231,212.331,-62.311,-177.836,7.184,148.715
C08244=1163.225,212.579,-62.335,-177.833,7.186,148.715
C08245=1163.222,212.829,-62.360,-177.830,7.189,148.715
C08246=1163.217,213.077,-62.385,-177.828,7.191,148.714
C08247=1163.212,213.326,-62.410,-177.825,7.194,148.714
C08248=1163.208,213.574,-62.434,-177.823,7.196,148.714
C08249=1163.203,213.823,-62.460,-177.819,7.198,148.714
C08250=1163.199,214.072,-62.484,-177.817,7.201,148.714
C08251=1163.194,214.320,-62.509,-177.814,7.203,148.713
C08252=1163.190,214.569,-62.535,-177.812,7.205,148.713
C08253=1163.185,214.818,-62.559,-177.808,7.208,148.713
C08254=1163.181,215.067,-62.584,-177.806,7.210,148.713
C08255=1163.176,215.315,-62.609,-177.803,7.213,148.712
C08256=1163.172,215.565,-62.634,-177.801,7.215,148.712
C08257=1163.168,215.812,-62.659,-177.798,7.218,148.712
C08258=1163.163,216.062,-62.684,-177.795,7.219,148.712
C08259=1163.158,216.311,-62.709,-177.793,7.222,148.712
C08260=1163.154,216.559,-62.734,-177.789,7.225,148.711
C08261=1163.149,216.808,-62.758,-177.787,7.227,148.711
C08262=1163.145,217.057,-62.784,-177.784,7.230,148.711
C08263=1163.140,217.305,-62.809,-177.782,7.232,148.711
C08264=1163.136,217.554,-62.835,-177.778,7.234,148.711
C08265=1163.131,217.802,-62.859,-177.776,7.237,148.710
C08266=1163.127,218.051,-62.884,-177.773,7.239,148.710
C08267=1163.122,218.299,-62.910,-177.771,7.241,148.710
C08268=1163.118,218.549,-62.935,-177.768,7.244,148.710
C08269=1163.113,218.797,-62.960,-177.765,7.246,148.710
C08270=1163.108,219.046,-62.985,-177.763,7.249,148.710
C08271=1163.104,219.294,-63.010,-177.760,7.251,148.709
C08272=1163.100,219.544,-63.035,-177.757,7.254,148.709
C08273=1163.096,219.792,-63.061,-177.754,7.256,148.709
C08274=1163.091,220.040,-63.086,-177.752,7.258,148.709
C08275=1163.086,220.290,-63.111,-177.748,7.261,148.708
C08276=1163.081,220.538,-63.137,-177.746,7.263,148.708
C08277=1163.077,220.787,-63.162,-177.743,7.266,148.708
C08278=1163.073,221.035,-63.187,-177.741,7.268,148.708
C08279=1163.068,221.284,-63.212,-177.738,7.271,148.708
C08280=1163.064,221.533,-63.238,-177.735,7.273,148.707
C08281=1163.059,221.781,-63.263,-177.733,7.275,148.707
C08282=1163.055,222.030,-63.288,-177.729,7.278,148.707
C08283=1163.050,222.278,-63.314,-177.727,7.280,148.707
C08284=1163.046,222.527,-63.340,-177.724,7.283,148.707
C08285=1163.042,222.776,-63.365,-177.722,7.285,148.707
C08286=1163.036,223.025,-63.390,-177.719,7.288,148.706
C08287=1163.032,223.274,-63.416,-177.716,7.290,148.706
C08288=1163.027,223.522,-63.441,-177.713,7.293,148.706
C08289=1163.023,223.771,-63.467,-177.711,7.295,148.706
C08290=1163.019,224.019,-63.493,-177.708,7.297,148.706
C08291=1163.014,224.268,-63.517,-177.705,7.300,148.706
C08292=1163.010,224.517,-63.543,-177.703,7.302,148.705
C08293=1163.005,224.766,-63.569,-177.700,7.305,148.705
C08294=1163.001,225.014,-63.594,-177.697,7.308,148.705
C08295=1162.996,225.263,-63.620,-177.694,7.310,148.705
C08296=1162.992,225.511,-63.646,-177.692,7.313,148.705
C08297=1162.987,225.759,-63.671,-177.689,7.315,148.704
C08298=1162.983,226.008,-63.697,-177.686,7.317,148.704
C08299=1162.979,226.257,-63.723,-177.683,7.320,148.704
C08300=1162.974,226.505,-63.748,-177.681,7.322,148.704
C08301=1162.970,226.754,-63.774,-177.678,7.325,148.704
C08302=1162.965,227.003,-63.800,-177.675,7.328,148.704
C08303=1162.961,227.252,-63.826,-177.673,7.330,148.703
C08304=1162.956,227.500,-63.851,-177.670,7.333,148.703
C08305=1162.952,227.749,-63.877,-177.668,7.335,148.703
C08306=1162.947,227.998,-63.903,-177.664,7.337,148.703
C08307=1162.943,228.246,-63.928,-177.662,7.340,148.703
C08308=1162.938,228.495,-63.954,-177.659,7.342,148.703
C08309=1162.934,228.743,-63.980,-177.656,7.345,148.702
C08310=1162.929,228.992,-64.006,-177.654,7.347,148.702
C08311=1162.924,229.241,-64.031,-177.651,7.350,148.702
C08312=1162.920,229.489,-64.057,-177.648,7.353,148.702
C08313=1162.916,229.738,-64.083,-177.646,7.355,148.702
C08314=1162.912,229.987,-64.109,-177.643,7.357,148.701
C08315=1162.907,230.235,-64.136,-177.640,7.360,148.701
C08316=1162.902,230.484,-64.161,-177.638,7.363,148.701
C08317=1162.898,230.732,-64.187,-177.634,7.365,148.701
C08318=1162.894,230.981,-64.213,-177.632,7.368,148.701
C08319=1162.889,231.230,-64.239,-177.629,7.370,148.701
C08320=1162.884,231.478,-64.265,-177.626,7.373,148.700
C08321=1162.880,231.727,-64.291,-177.623,7.376,148.700
C08322=1162.876,231.975,-64.316,-177.621,7.378,148.700
C08323=1162.871,232.224,-64.343,-177.618,7.381,148.700
C08324=1162.867,232.473,-64.369,-177.616,7.383,148.700
C08325=1162.863,232.721,-64.395,-177.613,7.386,148.700
C08326=1162.858,232.970,-64.420,-177.610,7.388,148.700
C08327=1162.853,233.219,-64.447,-177.608,7.390,148.699
C08328=1162.849,233.467,-64.473,-177.605,7.393,148.699
C08329=1162.845,233.716,-64.499,-177.602,7.396,148.699
C08330=1162.840,233.965,-64.525,-177.599,7.398,148.699
C08331=1162.836,234.213,-64.552,-177.597,7.401,148.699
C08332=1162.831,234.461,-64.577,-177.594,7.404,148.699
C08333=1162.826,234.710,-64.604,-177.592,7.406,148.699
C08334=1162.822,234.958,-64.630,-177.588,7.409,148.698
C08335=1162.817,235.208,-64.656,-177.586,7.411,148.698
C08336=1162.813,235.456,-64.683,-177.583,7.414,148.698
C08337=1162.809,235.728,-64.711,-177.580,7.416,148.698
C08338=1162.803,235.999,-64.740,-177.577,7.420,148.698
C08339=1162.799,236.271,-64.768,-177.574,7.423,148.697
C08340=1162.794,236.543,-64.798,-177.571,7.426,148.697
C08341=1162.789,236.791,-64.823,-177.569,7.428,148.697
C08342=1162.785,237.040,-64.850,-177.566,7.431,148.697
C08343=1162.780,237.289,-64.876,-177.563,7.433,148.697
C08344=1162.777,237.537,-64.903,-177.560,7.435,148.697
C08345=1162.772,237.785,-64.930,-177.558,7.438,148.697
C08346=1162.768,238.034,-64.955,-177.554,7.441,148.696
C08347=1162.762,238.282,-64.982,-177.552,7.443,148.696
C08348=1162.758,238.531,-65.008,-177.549,7.446,148.696
C08349=1162.754,238.779,-65.035,-177.547,7.449,148.696
C08350=1162.749,239.028,-65.061,-177.544,7.451,148.696
C08351=1162.745,239.277,-65.088,-177.541,7.454,148.696
C08352=1162.741,239.525,-65.114,-177.538,7.457,148.696
C08353=1162.736,239.774,-65.141,-177.536,7.460,148.696
C08354=1162.731,240.022,-65.168,-177.534,7.462,148.696
C08355=1162.727,240.271,-65.194,-177.530,7.464,148.695
C08356=1162.722,240.520,-65.220,-177.528,7.467,148.695
C08357=1162.718,240.768,-65.247,-177.525,7.469,148.695
C08358=1162.714,241.016,-65.274,-177.523,7.472,148.695
C08359=1162.709,241.265,-65.300,-177.519,7.475,148.695
C08360=1162.705,241.514,-65.327,-177.517,7.478,148.695
C08361=1162.700,241.762,-65.354,-177.514,7.480,148.695
C08362=1162.696,242.010,-65.380,-177.512,7.483,148.694
C08363=1162.691,242.260,-65.407,-177.509,7.486,148.694
C08364=1162.687,242.508,-65.433,-177.506,7.489,148.694
C08365=1162.683,242.756,-65.460,-177.503,7.491,148.694
C08366=1162.678,243.005,-65.487,-177.501,7.494,148.694
C08367=1162.674,243.253,-65.514,-177.498,7.497,148.694
C08368=1162.669,243.502,-65.540,-177.496,7.499,148.694
C08369=1162.664,243.751,-65.567,-177.492,7.501,148.693
C08370=1162.661,243.999,-65.594,-177.490,7.504,148.693
C08371=1162.657,244.248,-65.621,-177.487,7.507,148.693
C08372=1162.652,244.496,-65.648,-177.485,7.509,148.693
C08373=1162.648,244.745,-65.675,-177.482,7.512,148.693
C08374=1162.643,244.993,-65.702,-177.479,7.515,148.693
C08375=1162.639,245.242,-65.729,-177.476,7.518,148.693
C08376=1162.635,245.490,-65.755,-177.474,7.520,148.693
C08377=1162.630,245.738,-65.782,-177.471,7.523,148.693
C08378=1162.625,245.987,-65.809,-177.468,7.526,148.693
C08379=1162.621,246.235,-65.836,-177.465,7.529,148.692
C08380=1162.617,246.484,-65.862,-177.463,7.531,148.692
C08381=1162.612,246.733,-65.889,-177.460,7.534,148.692
C08382=1162.608,246.981,-65.917,-177.457,7.536,148.692
C08383=1162.603,247.230,-65.944,-177.455,7.539,148.692
C08384=1162.599,247.478,-65.971,-177.452,7.542,148.692
C08385=1162.595,247.726,-65.998,-177.450,7.544,148.692
C08386=1162.590,247.975,-66.025,-177.446,7.547,148.691
C08387=1162.586,248.223,-66.052,-177.444,7.550,148.691
C08388=1162.581,248.472,-66.079,-177.441,7.552,148.691
C08389=1162.577,248.721,-66.106,-177.439,7.555,148.691
C08390=1162.573,248.969,-66.133,-177.436,7.558,148.691
C08391=1162.568,249.218,-66.160,-177.433,7.561,148.691
C08392=1162.564,249.466,-66.187,-177.430,7.564,148.691
C08393=1162.559,249.714,-66.215,-177.428,7.566,148.691
C08394=1162.555,249.963,-66.242,-177.425,7.569,148.691
C08395=1162.551,250.212,-66.269,-177.422,7.572,148.691
C08396=1162.546,250.460,-66.296,-177.419,7.575,148.691
C08397=1162.541,250.709,-66.323,-177.417,7.577,148.690
C08398=1162.538,250.956,-66.351,-177.414,7.580,148.690
C08399=1162.534,251.205,-66.378,-177.412,7.583,148.690
C08400=1162.529,251.454,-66.405,-177.409,7.586,148.690
C08401=1162.524,251.702,-66.432,-177.406,7.588,148.690
C08402=1162.520,251.950,-66.460,-177.403,7.590,148.690
C08403=1162.515,252.199,-66.487,-177.401,7.593,148.690
C08404=1162.511,252.448,-66.514,-177.398,7.596,148.690
C08405=1162.507,252.697,-66.542,-177.395,7.599,148.690
C08406=1162.502,252.944,-66.569,-177.392,7.602,148.690
C08407=1162.498,253.193,-66.596,-177.390,7.604,148.690
C08408=1162.493,253.442,-66.624,-177.387,7.607,148.689
C08409=1162.489,253.690,-66.652,-177.385,7.610,148.689
C08410=1162.484,253.938,-66.679,-177.382,7.613,148.689
C08411=1162.480,254.186,-66.706,-177.379,7.616,148.689
C08412=1162.476,254.436,-66.734,-177.377,7.618,148.689
C08413=1162.471,254.684,-66.761,-177.374,7.621,148.689
C08414=1162.467,254.932,-66.789,-177.371,7.624,148.689
C08415=1162.463,255.181,-66.816,-177.368,7.627,148.689
C08416=1162.459,255.429,-66.844,-177.365,7.630,148.689
C08417=1162.454,255.677,-66.871,-177.363,7.632,148.689
C08418=1162.450,255.926,-66.899,-177.361,7.635,148.689
C08419=1162.445,256.175,-66.927,-177.358,7.638,148.688
C08420=1162.440,256.423,-66.954,-177.355,7.641,148.688
C08421=1162.436,256.671,-66.982,-177.352,7.644,148.688
C08422=1162.432,256.920,-67.010,-177.349,7.647,148.688
C08423=1162.427,257.168,-67.037,-177.347,7.649,148.688
C08424=1162.424,257.417,-67.065,-177.345,7.652,148.688
C08425=1162.419,257.665,-67.092,-177.342,7.655,148.688
C08426=1162.415,257.913,-67.120,-177.339,7.658,148.688
C08427=1162.410,258.162,-67.148,-177.336,7.661,148.688
C08428=1162.406,258.411,-67.176,-177.333,7.663,148.688
C08429=1162.401,258.659,-67.203,-177.331,7.666,148.688
C08430=1162.397,258.907,-67.231,-177.329,7.669,148.688
C08431=1162.393,259.156,-67.259,-177.325,7.671,148.687
C08432=1162.388,259.403,-67.286,-177.323,7.674,148.687
C08433=1162.384,259.652,-67.315,-177.320,7.677,148.687
C08434=1162.379,259.901,-67.342,-177.317,7.680,148.687
C08435=1162.376,260.149,-67.370,-177.315,7.682,148.687
C08436=1162.371,260.397,-67.398,-177.312,7.685,148.687
C08437=1162.366,260.646,-67.426,-177.309,7.688,148.687
C08438=1162.362,260.895,-67.454,-177.307,7.691,148.687
C08439=1162.358,261.143,-67.482,-177.304,7.694,148.687
C08440=1162.354,261.391,-67.510,-177.301,7.697,148.687
C08441=1162.349,261.664,-67.540,-177.298,7.700,148.687
C08442=1162.344,261.937,-67.571,-177.296,7.703,148.687
C08443=1162.339,262.211,-67.602,-177.293,7.706,148.687
C08444=1162.334,262.484,-67.633,-177.289,7.710,148.687
C08445=1162.330,262.733,-67.661,-177.287,7.713,148.687
C08446=1162.326,262.981,-67.689,-177.284,7.715,148.687
C08447=1162.321,263.229,-67.717,-177.282,7.718,148.687
C08448=1162.317,263.477,-67.745,-177.279,7.721,148.686
C08449=1162.312,263.726,-67.772,-177.276,7.723,148.686
C08450=1162.308,263.975,-67.801,-177.273,7.726,148.686
C08451=1162.304,264.223,-67.829,-177.271,7.729,148.686
C08452=1162.300,264.471,-67.857,-177.268,7.732,148.686
C08453=1162.295,264.719,-67.885,-177.266,7.734,148.686
C08454=1162.291,264.968,-67.913,-177.263,7.737,148.686
C08455=1162.286,265.216,-67.942,-177.260,7.740,148.686
C08456=1162.282,265.465,-67.970,-177.257,7.743,148.686
C08457=1162.277,265.713,-67.998,-177.255,7.746,148.686
C08458=1162.273,265.961,-68.026,-177.252,7.749,148.686
C08459=1162.269,266.209,-68.054,-177.249,7.752,148.686
C08460=1162.264,266.458,-68.083,-177.247,7.756,148.686
C08461=1162.261,266.707,-68.111,-177.244,7.758,148.686
C08462=1162.256,266.955,-68.139,-177.242,7.761,148.686
C08463=1162.252,267.204,-68.168,-177.239,7.764,148.686
C08464=1162.247,267.452,-68.196,-177.236,7.766,148.686
C08465=1162.243,267.700,-68.225,-177.234,7.769,148.686
C08466=1162.238,267.948,-68.253,-177.231,7.772,148.686
C08467=1162.234,268.196,-68.281,-177.228,7.775,148.686
C08468=1162.229,268.445,-68.310,-177.225,7.778,148.686
C08469=1162.226,268.693,-68.338,-177.223,7.781,148.685
C08470=1162.221,268.942,-68.367,-177.220,7.784,148.685
C08471=1162.217,269.190,-68.394,-177.218,7.786,148.685
C08472=1162.213,269.438,-68.424,-177.215,7.789,148.685
C08473=1162.208,269.686,-68.452,-177.213,7.793,148.685
C08474=1162.204,269.935,-68.480,-177.210,7.796,148.685
C08475=1162.199,270.184,-68.509,-177.207,7.799,148.685
C08476=1162.195,270.431,-68.538,-177.204,7.801,148.685
C08477=1162.191,270.680,-68.566,-177.202,7.804,148.685
C08478=1162.186,270.928,-68.594,-177.199,7.807,148.685
C08479=1162.182,271.177,-68.623,-177.196,7.810,148.685
C08480=1162.178,271.425,-68.652,-177.193,7.813,148.685
C08481=1162.173,271.673,-68.680,-177.191,7.816,148.685
C08482=1162.169,271.922,-68.709,-177.188,7.818,148.685
C08483=1162.165,272.170,-68.738,-177.186,7.822,148.685
C08484=1162.160,272.418,-68.766,-177.183,7.825,148.685
C08485=1162.156,272.667,-68.795,-177.181,7.828,148.685
C08486=1162.152,272.915,-68.824,-177.178,7.831,148.685
C08487=1162.147,273.163,-68.852,-177.175,7.833,148.685
C08488=1162.143,273.411,-68.881,-177.172,7.836,148.685
C08489=1162.139,273.660,-68.910,-177.169,7.839,148.685
C08490=1162.135,273.907,-68.939,-177.167,7.843,148.685
C08491=1162.130,274.156,-68.967,-177.164,7.846,148.685
C08492=1162.126,274.405,-68.996,-177.162,7.849,148.685
C08493=1162.122,274.652,-69.025,-177.159,7.852,148.685
C08494=1162.117,274.901,-69.053,-177.156,7.855,148.685
C08495=1162.113,275.150,-69.083,-177.153,7.857,148.685
C08496=1162.109,275.398,-69.111,-177.151,7.860,148.685
C08497=1162.104,275.646,-69.140,-177.149,7.863,148.685
C08498=1162.100,275.894,-69.169,-177.146,7.866,148.685
C08499=1162.096,276.143,-69.198,-177.143,7.869,148.685
C08500=1162.092,276.391,-69.228,-177.141,7.872,148.685
C08501=1162.087,276.639,-69.255,-177.138,7.875,148.685
C08502=1162.083,276.887,-69.285,-177.135,7.878,148.685
C08503=1162.079,277.136,-69.314,-177.133,7.881,148.685
C08504=1162.074,277.384,-69.343,-177.130,7.884,148.685
C08505=1162.070,277.632,-69.372,-177.127,7.887,148.685
C08506=1162.066,277.881,-69.400,-177.125,7.890,148.685
C08507=1162.062,278.129,-69.430,-177.122,7.893,148.685
C08508=1162.057,278.377,-69.459,-177.120,7.896,148.685
C08509=1162.053,278.626,-69.488,-177.117,7.899,148.685
C08510=1162.048,278.874,-69.517,-177.114,7.902,148.685
C08511=1162.044,279.122,-69.546,-177.111,7.905,148.685
C08512=1162.040,279.370,-69.576,-177.108,7.908,148.685
C08513=1162.036,279.619,-69.604,-177.106,7.911,148.685
C08514=1162.032,279.867,-69.634,-177.103,7.914,148.685
C08515=1162.027,280.114,-69.663,-177.101,7.917,148.685
C08516=1162.023,280.363,-69.692,-177.098,7.920,148.685
C08517=1162.018,280.612,-69.721,-177.096,7.922,148.685
C08518=1162.014,280.860,-69.750,-177.093,7.925,148.685
C08519=1162.010,281.108,-69.780,-177.091,7.928,148.685
C08520=1162.006,281.356,-69.809,-177.088,7.931,148.685
C08521=1162.001,281.604,-69.838,-177.085,7.934,148.685
C08522=1161.997,281.852,-69.868,-177.082,7.937,148.685
C08523=1161.993,282.101,-69.897,-177.080,7.941,148.685
C08524=1161.988,282.349,-69.926,-177.077,7.944,148.685
C08525=1161.984,282.598,-69.955,-177.075,7.947,148.685
C08526=1161.980,282.846,-69.985,-177.072,7.949,148.685
C08527=1161.976,283.094,-70.014,-177.070,7.953,148.685
C08528=1161.972,283.343,-70.044,-177.067,7.956,148.685
C08529=1161.967,283.590,-70.073,-177.064,7.959,148.685
C08530=1161.963,283.838,-70.102,-177.061,7.962,148.685
C08531=1161.958,284.087,-70.132,-177.059,7.965,148.685
C08532=1161.954,284.335,-70.161,-177.056,7.968,148.685
C08533=1161.950,284.583,-70.191,-177.053,7.971,148.685
C08534=1161.946,284.831,-70.220,-177.051,7.974,148.685
C08535=1161.942,285.080,-70.250,-177.048,7.977,148.685
C08536=1161.937,285.328,-70.280,-177.046,7.980,148.685
C08537=1161.933,285.577,-70.309,-177.043,7.983,148.685
C08538=1161.928,285.825,-70.338,-177.041,7.986,148.685
C08539=1161.924,286.073,-70.368,-177.038,7.989,148.685
C08540=1161.920,286.321,-70.398,-177.035,7.992,148.685
C08541=1161.916,286.569,-70.428,-177.032,7.995,148.685
C08542=1161.912,286.817,-70.457,-177.030,7.998,148.685
C08543=1161.907,287.065,-70.486,-177.027,8.001,148.685
C08544=1161.902,287.313,-70.516,-177.025,8.004,148.685
C08545=1161.898,287.588,-70.549,-177.021,8.008,148.685
C08546=1161.893,287.863,-70.581,-177.019,8.011,148.685
C08547=1161.889,288.138,-70.615,-177.016,8.014,148.685
C08548=1161.884,288.413,-70.647,-177.013,8.018,148.685
C08549=1161.880,288.662,-70.677,-177.010,8.021,148.685
C08550=1161.875,288.910,-70.708,-177.008,8.024,148.685
C08551=1161.871,289.158,-70.737,-177.005,8.027,148.685
C08552=1161.867,289.406,-70.767,-177.002,8.030,148.685
C08553=1161.863,289.655,-70.796,-177.000,8.034,148.685
C08554=1161.858,289.903,-70.827,-176.997,8.037,148.685
C08555=1161.854,290.151,-70.857,-176.994,8.040,148.685
C08556=1161.850,290.400,-70.886,-176.992,8.043,148.685
C08557=1161.846,290.647,-70.916,-176.989,8.046,148.685
C08558=1161.841,290.896,-70.946,-176.987,8.049,148.685
C08559=1161.837,291.144,-70.976,-176.984,8.052,148.685
C08560=1161.833,291.392,-71.006,-176.982,8.055,148.685
C08561=1161.828,291.640,-71.036,-176.979,8.058,148.685
C08562=1161.824,291.888,-71.066,-176.977,8.061,148.686
C08563=1161.820,292.136,-71.096,-176.974,8.064,148.686
C08564=1161.816,292.384,-71.126,-176.971,8.067,148.686
C08565=1161.811,292.632,-71.156,-176.969,8.070,148.686
C08566=1161.807,292.881,-71.185,-176.966,8.073,148.686
C08567=1161.803,293.129,-71.216,-176.963,8.076,148.686
C08568=1161.799,293.378,-71.246,-176.961,8.080,148.686
C08569=1161.795,293.625,-71.276,-176.958,8.083,148.686
C08570=1161.790,293.874,-71.306,-176.955,8.087,148.686
C08571=1161.786,294.122,-71.336,-176.953,8.090,148.686
C08572=1161.782,294.369,-71.367,-176.950,8.093,148.686
C08573=1161.778,294.618,-71.396,-176.947,8.096,148.686
C08574=1161.774,294.865,-71.427,-176.945,8.099,148.686
C08575=1161.769,295.114,-71.457,-176.942,8.102,148.686
C08576=1161.766,295.362,-71.487,-176.940,8.105,148.686
C08577=1161.761,295.610,-71.518,-176.937,8.108,148.686
C08578=1161.757,295.859,-71.547,-176.935,8.111,148.686
C08579=1161.752,296.107,-71.578,-176.932,8.114,148.686
C08580=1161.748,296.355,-71.608,-176.929,8.117,148.686
C08581=1161.743,296.603,-71.638,-176.927,8.121,148.686
C08582=1161.740,296.851,-71.669,-176.924,8.124,148.686
C08583=1161.735,297.099,-71.700,-176.922,8.127,148.687
C08584=1161.731,297.347,-71.729,-176.919,8.130,148.687
C08585=1161.727,297.595,-71.760,-176.916,8.133,148.687
C08586=1161.723,297.843,-71.790,-176.914,8.136,148.687
C08587=1161.718,298.092,-71.820,-176.911,8.139,148.687
C08588=1161.715,298.340,-71.851,-176.908,8.143,148.687
C08589=1161.710,298.588,-71.881,-176.906,8.146,148.687
C08590=1161.706,298.835,-71.912,-176.903,8.149,148.687
C08591=1161.702,299.083,-71.942,-176.901,8.152,148.687
C08592=1161.697,299.333,-71.973,-176.898,8.155,148.687
C08593=1161.693,299.580,-72.003,-176.895,8.159,148.687
C08594=1161.689,299.828,-72.034,-176.893,8.162,148.687
C08595=1161.685,300.076,-72.064,-176.890,8.165,148.687
C08596=1161.681,300.325,-72.095,-176.888,8.168,148.687
C08597=1161.676,300.573,-72.126,-176.885,8.171,148.688
C08598=1161.672,300.820,-72.156,-176.883,8.174,148.687
C08599=1161.667,301.069,-72.186,-176.880,8.177,148.687
C08600=1161.663,301.317,-72.217,-176.878,8.180,148.688
C08601=1161.660,301.565,-72.247,-176.874,8.184,148.688
C08602=1161.655,301.813,-72.278,-176.872,8.187,148.688
C08603=1161.651,302.062,-72.309,-176.869,8.190,148.688
C08604=1161.647,302.309,-72.339,-176.867,8.194,148.688
C08605=1161.642,302.557,-72.370,-176.864,8.197,148.688
C08606=1161.638,302.805,-72.401,-176.862,8.200,148.688
C08607=1161.635,303.054,-72.431,-176.859,8.203,148.688
C08608=1161.630,303.302,-72.462,-176.857,8.206,148.688
C08609=1161.625,303.550,-72.493,-176.854,8.209,148.688
C08610=1161.621,303.798,-72.524,-176.852,8.212,148.688
C08611=1161.617,304.046,-72.554,-176.849,8.215,148.688
C08612=1161.613,304.293,-72.586,-176.846,8.220,148.689
C08613=1161.609,304.542,-72.617,-176.843,8.222,148.689
C08614=1161.604,304.790,-72.648,-176.841,8.226,148.689
C08615=1161.600,305.038,-72.678,-176.838,8.229,148.689
C08616=1161.597,305.286,-72.709,-176.836,8.232,148.689
C08617=1161.592,305.534,-72.740,-176.833,8.235,148.689
C08618=1161.587,305.782,-72.770,-176.831,8.238,148.689
C08619=1161.584,306.030,-72.802,-176.828,8.241,148.689
C08620=1161.579,306.278,-72.833,-176.826,8.245,148.689
C08621=1161.574,306.526,-72.864,-176.823,8.248,148.689
C08622=1161.571,306.774,-72.894,-176.820,8.252,148.690
C08623=1161.567,307.022,-72.925,-176.818,8.255,148.689
C08624=1161.563,307.270,-72.957,-176.815,8.258,148.690
C08625=1161.558,307.518,-72.988,-176.812,8.261,148.690
C08626=1161.554,307.766,-73.018,-176.810,8.264,148.690
C08627=1161.550,308.014,-73.050,-176.807,8.267,148.690
C08628=1161.545,308.262,-73.081,-176.805,8.270,148.690
C08629=1161.541,308.511,-73.112,-176.802,8.274,148.690
C08630=1161.537,308.758,-73.144,-176.800,8.277,148.690
C08631=1161.534,309.007,-73.174,-176.797,8.281,148.690
C08632=1161.529,309.255,-73.205,-176.794,8.284,148.690
C08633=1161.525,309.502,-73.236,-176.792,8.287,148.691
C08634=1161.521,309.751,-73.268,-176.789,8.290,148.691
C08635=1161.516,309.998,-73.298,-176.787,8.293,148.691
C08636=1161.512,310.247,-73.330,-176.784,8.296,148.691
C08637=1161.508,310.494,-73.361,-176.781,8.300,148.691
C08638=1161.504,310.743,-73.393,-176.779,8.303,148.691
C08639=1161.499,310.990,-73.424,-176.776,8.307,148.691
C08640=1161.496,311.239,-73.455,-176.774,8.310,148.691
C08641=1161.491,311.486,-73.486,-176.771,8.313,148.691
C08642=1161.487,311.735,-73.518,-176.769,8.316,148.691
C08643=1161.483,311.982,-73.549,-176.766,8.319,148.691
C08644=1161.479,312.231,-73.581,-176.763,8.323,148.692
C08645=1161.475,312.478,-73.611,-176.761,8.326,148.692
C08646=1161.471,312.726,-73.643,-176.758,8.329,148.692
C08647=1161.466,312.974,-73.674,-176.756,8.333,148.692
C08648=1161.462,313.223,-73.706,-176.753,8.336,148.692
C08649=1161.458,313.499,-73.741,-176.751,8.340,148.692
C08650=1161.453,313.777,-73.776,-176.748,8.343,148.692
C08651=1161.448,314.054,-73.811,-176.745,8.347,148.692
C08652=1161.443,314.331,-73.846,-176.742,8.351,148.693
C08653=1161.439,314.579,-73.878,-176.739,8.354,148.693
C08654=1161.435,314.827,-73.909,-176.737,8.357,148.693
C08655=1161.431,315.075,-73.941,-176.734,8.360,148.693
C08656=1161.427,315.323,-73.973,-176.732,8.363,148.693
C08657=1161.422,315.571,-74.005,-176.729,8.368,148.693
C08658=1161.418,315.819,-74.036,-176.726,8.371,148.693
C08659=1161.414,316.067,-74.067,-176.724,8.374,148.693
C08660=1161.410,316.315,-74.099,-176.722,8.377,148.694
C08661=1161.407,316.563,-74.131,-176.719,8.380,148.694
C08662=1161.401,316.811,-74.162,-176.717,8.383,148.694
C08663=1161.398,317.059,-74.194,-176.714,8.387,148.694
C08664=1161.393,317.307,-74.226,-176.711,8.390,148.694
C08665=1161.390,317.555,-74.258,-176.709,8.394,148.694
C08666=1161.386,317.803,-74.289,-176.706,8.397,148.694
C08667=1161.380,318.051,-74.321,-176.704,8.400,148.694
C08668=1161.377,318.299,-74.353,-176.701,8.403,148.695
C08669=1161.373,318.547,-74.385,-176.698,8.407,148.695
C08670=1161.369,318.794,-74.416,-176.696,8.410,148.695
C08671=1161.364,319.043,-74.448,-176.693,8.414,148.695
C08672=1161.361,319.291,-74.480,-176.691,8.417,148.695
C08673=1161.356,319.538,-74.512,-176.688,8.420,148.695
C08674=1161.352,319.786,-74.544,-176.686,8.424,148.695
C08675=1161.348,320.034,-74.576,-176.683,8.427,148.696
C08676=1161.344,320.282,-74.608,-176.680,8.430,148.696
C08677=1161.339,320.530,-74.640,-176.678,8.434,148.696
C08678=1161.336,320.778,-74.672,-176.676,8.437,148.696
C08679=1161.331,321.025,-74.703,-176.673,8.441,148.696
C08680=1161.327,321.274,-74.736,-176.670,8.444,148.696
C08681=1161.323,321.522,-74.768,-176.668,8.447,148.696
C08682=1161.319,321.769,-74.799,-176.666,8.450,148.697
C08683=1161.315,322.018,-74.831,-176.663,8.453,148.697
C08684=1161.311,322.266,-74.863,-176.660,8.458,148.697
C08685=1161.307,322.514,-74.895,-176.658,8.461,148.697
C08686=1161.302,322.761,-74.927,-176.655,8.464,148.697
C08687=1161.299,323.009,-74.960,-176.653,8.467,148.697
C08688=1161.294,323.257,-74.992,-176.650,8.470,148.697
C08689=1161.290,323.505,-75.024,-176.647,8.474,148.698
C08690=1161.286,323.752,-75.056,-176.645,8.477,148.698
C08691=1161.282,324.001,-75.088,-176.642,8.481,148.698
C08692=1161.278,324.249,-75.120,-176.640,8.484,148.698
C08693=1161.274,324.497,-75.153,-176.638,8.487,148.698
C08694=1161.270,324.744,-75.185,-176.635,8.491,148.698
C08695=1161.265,324.992,-75.217,-176.632,8.494,148.698
C08696=1161.261,325.240,-75.249,-176.630,8.498,148.699
C08697=1161.257,325.488,-75.282,-176.628,8.501,148.699
C08698=1161.254,325.736,-75.314,-176.624,8.505,148.699
C08699=1161.249,325.984,-75.346,-176.622,8.508,148.699
C08700=1161.245,326.231,-75.378,-176.620,8.511,148.699
C08701=1161.241,326.479,-75.411,-176.617,8.515,148.699
C08702=1161.237,326.728,-75.443,-176.615,8.518,148.699
C08703=1161.233,326.975,-75.476,-176.612,8.522,148.700
C08704=1161.229,327.223,-75.507,-176.609,8.525,148.700
C08705=1161.224,327.471,-75.540,-176.607,8.528,148.700
C08706=1161.220,327.719,-75.573,-176.605,8.532,148.700
C08707=1161.216,327.967,-75.605,-176.602,8.535,148.700
C08708=1161.212,328.214,-75.638,-176.599,8.539,148.701
C08709=1161.208,328.462,-75.670,-176.597,8.542,148.701
C08710=1161.204,328.711,-75.702,-176.595,8.545,148.701
C08711=1161.199,328.958,-75.735,-176.592,8.549,148.701
C08712=1161.196,329.206,-75.767,-176.589,8.552,148.701
C08713=1161.191,329.454,-75.800,-176.587,8.556,148.701
C08714=1161.187,329.702,-75.832,-176.584,8.559,148.702
C08715=1161.184,329.949,-75.865,-176.582,8.563,148.702
C08716=1161.179,330.198,-75.897,-176.579,8.566,148.702
C08717=1161.175,330.445,-75.931,-176.577,8.570,148.702
C08718=1161.172,330.693,-75.963,-176.574,8.572,148.702
C08719=1161.167,330.941,-75.995,-176.571,8.577,148.702
C08720=1161.162,331.188,-76.028,-176.569,8.580,148.703
C08721=1161.159,331.436,-76.060,-176.567,8.583,148.703
C08722=1161.155,331.684,-76.093,-176.564,8.586,148.703
C08723=1161.150,331.932,-76.127,-176.562,8.591,148.703
C08724=1161.146,332.180,-76.159,-176.559,8.594,148.703
C08725=1161.143,332.428,-76.192,-176.556,8.597,148.703
C08726=1161.138,332.675,-76.225,-176.554,8.600,148.704
C08727=1161.134,332.924,-76.257,-176.551,8.604,148.704
C08728=1161.130,333.171,-76.290,-176.549,8.607,148.704
C08729=1161.126,333.419,-76.323,-176.547,8.611,148.704
C08730=1161.122,333.667,-76.355,-176.544,8.615,148.705
C08731=1161.118,333.915,-76.388,-176.542,8.618,148.705
C08732=1161.114,334.163,-76.422,-176.539,8.621,148.705
C08733=1161.110,334.410,-76.455,-176.536,8.624,148.705
C08734=1161.106,334.658,-76.487,-176.534,8.629,148.705
C08735=1161.102,334.906,-76.520,-176.531,8.632,148.705
C08736=1161.098,335.154,-76.553,-176.529,8.635,148.706
C08737=1161.093,335.402,-76.586,-176.526,8.639,148.706
C08738=1161.089,335.649,-76.619,-176.524,8.643,148.706
C08739=1161.085,335.897,-76.652,-176.522,8.646,148.706
C08740=1161.081,336.145,-76.685,-176.519,8.649,148.707
C08741=1161.077,336.393,-76.717,-176.516,8.653,148.707
C08742=1161.073,336.640,-76.751,-176.514,8.656,148.707
C08743=1161.069,336.888,-76.784,-176.512,8.660,148.707
C08744=1161.065,337.136,-76.817,-176.508,8.664,148.707
C08745=1161.061,337.384,-76.850,-176.506,8.667,148.707
C08746=1161.057,337.631,-76.883,-176.504,8.670,148.708
C08747=1161.053,337.879,-76.916,-176.502,8.673,148.708
C08748=1161.048,338.127,-76.950,-176.499,8.678,148.708
C08749=1161.044,338.375,-76.983,-176.496,8.681,148.708
C08750=1161.040,338.622,-77.016,-176.494,8.684,148.708
C08751=1161.036,338.870,-77.049,-176.491,8.688,148.709
C08752=1161.032,339.118,-77.082,-176.489,8.691,148.709
C08753=1161.027,339.397,-77.120,-176.486,8.696,148.709
C08754=1161.023,339.677,-77.157,-176.483,8.700,148.709
C08755=1161.019,339.957,-77.195,-176.480,8.704,148.710
C08756=1161.014,340.237,-77.233,-176.477,8.708,148.710
C08757=1161.010,340.485,-77.266,-176.475,8.711,148.710
C08758=1161.006,340.732,-77.299,-176.473,8.714,148.710
C08759=1161.002,340.980,-77.332,-176.470,8.718,148.711
C08760=1160.997,341.228,-77.365,-176.468,8.722,148.711
C08761=1160.993,341.475,-77.398,-176.465,8.725,148.711
C08762=1160.990,341.723,-77.432,-176.463,8.728,148.711
C08763=1160.985,341.971,-77.466,-176.460,8.733,148.712
C08764=1160.981,342.219,-77.500,-176.458,8.736,148.712
C08765=1160.977,342.467,-77.533,-176.455,8.739,148.712
C08766=1160.973,342.714,-77.566,-176.453,8.743,148.712
C08767=1160.969,342.962,-77.600,-176.450,8.747,148.712
C08768=1160.965,343.209,-77.633,-176.447,8.751,148.713
C08769=1160.961,343.457,-77.666,-176.445,8.754,148.713
C08770=1160.957,343.705,-77.700,-176.443,8.757,148.713
C08771=1160.953,343.953,-77.734,-176.440,8.761,148.713
C08772=1160.948,344.201,-77.767,-176.438,8.765,148.714
C08773=1160.945,344.448,-77.801,-176.435,8.768,148.714
C08774=1160.940,344.695,-77.834,-176.432,8.772,148.714
C08775=1160.936,344.943,-77.867,-176.430,8.775,148.714
C08776=1160.932,345.191,-77.902,-176.428,8.779,148.715
C08777=1160.928,345.439,-77.935,-176.425,8.783,148.715
C08778=1160.924,345.687,-77.969,-176.423,8.786,148.715
C08779=1160.920,345.934,-78.002,-176.421,8.790,148.715
C08780=1160.915,346.182,-78.036,-176.418,8.794,148.716
C08781=1160.912,346.430,-78.070,-176.416,8.797,148.716
C08782=1160.908,346.677,-78.104,-176.413,8.800,148.716
C08783=1160.904,346.925,-78.137,-176.410,8.804,148.716
C08784=1160.899,347.173,-78.171,-176.408,8.808,148.716
C08785=1160.896,347.420,-78.205,-176.405,8.812,148.717
C08786=1160.892,347.668,-78.239,-176.403,8.815,148.717
C08787=1160.888,347.915,-78.272,-176.401,8.819,148.717
C08788=1160.883,348.163,-78.306,-176.398,8.823,148.718
C08789=1160.880,348.411,-78.340,-176.396,8.826,148.718
C08790=1160.876,348.658,-78.374,-176.394,8.829,148.718
C08791=1160.871,348.906,-78.408,-176.391,8.833,148.718
C08792=1160.868,349.154,-78.442,-176.388,8.837,148.718
C08793=1160.864,349.402,-78.475,-176.386,8.841,148.719
C08794=1160.859,349.649,-78.510,-176.384,8.844,148.719
C08795=1160.856,349.897,-78.544,-176.381,8.848,148.719
C08796=1160.851,350.145,-78.578,-176.378,8.852,148.720
C08797=1160.847,350.392,-78.612,-176.376,8.855,148.720
C08798=1160.844,350.639,-78.646,-176.373,8.859,148.720
C08799=1160.839,350.888,-78.680,-176.371,8.862,148.720
C08800=1160.835,351.135,-78.714,-176.369,8.866,148.720
C08801=1160.831,351.383,-78.748,-176.366,8.870,148.721
C08802=1160.828,351.630,-78.782,-176.364,8.873,148.721
C08803=1160.824,351.878,-78.815,-176.361,8.878,148.721
C08804=1160.820,352.126,-78.850,-176.359,8.881,148.722
C08805=1160.816,352.373,-78.884,-176.356,8.884,148.722
C08806=1160.811,352.621,-78.919,-176.354,8.889,148.722
C08807=1160.808,352.869,-78.953,-176.352,8.892,148.723
C08808=1160.803,353.117,-78.987,-176.349,8.896,148.723
C08809=1160.799,353.364,-79.020,-176.347,8.899,148.723
C08810=1160.795,353.612,-79.055,-176.344,8.904,148.723
C08811=1160.791,353.859,-79.089,-176.342,8.907,148.724
C08812=1160.787,354.107,-79.124,-176.339,8.910,148.724
C08813=1160.784,354.354,-79.158,-176.337,8.914,148.724
C08814=1160.779,354.602,-79.192,-176.334,8.918,148.724
C08815=1160.776,354.849,-79.227,-176.332,8.922,148.725
C08816=1160.771,355.097,-79.261,-176.330,8.925,148.725
C08817=1160.768,355.345,-79.295,-176.327,8.929,148.725
C08818=1160.763,355.592,-79.330,-176.324,8.933,148.726
C08819=1160.760,355.840,-79.365,-176.322,8.936,148.726
C08820=1160.756,356.087,-79.398,-176.320,8.940,148.726
C08821=1160.751,356.335,-79.433,-176.317,8.944,148.726
C08822=1160.748,356.582,-79.467,-176.315,8.948,148.727
C08823=1160.743,356.830,-79.502,-176.313,8.951,148.727
C08824=1160.739,357.078,-79.536,-176.310,8.956,148.727
C08825=1160.736,357.325,-79.570,-176.307,8.959,148.728
C08826=1160.732,357.573,-79.605,-176.305,8.963,148.728
C08827=1160.727,357.821,-79.640,-176.303,8.967,148.728
C08828=1160.724,358.068,-79.674,-176.300,8.971,148.729
C08829=1160.719,358.315,-79.709,-176.298,8.974,148.729
C08830=1160.716,358.563,-79.743,-176.295,8.978,148.729
C08831=1160.712,358.811,-79.778,-176.293,8.982,148.729
C08832=1160.708,359.059,-79.813,-176.291,8.985,148.730
C08833=1160.703,359.306,-79.847,-176.288,8.989,148.730
C08834=1160.700,359.554,-79.881,-176.286,8.993,148.730
C08835=1160.696,359.801,-79.916,-176.283,8.997,148.731
C08836=1160.692,360.049,-79.951,-176.280,9.001,148.731
C08837=1160.688,360.296,-79.985,-176.278,9.004,148.731
C08838=1160.684,360.544,-80.020,-176.276,9.009,148.732
C08839=1160.680,360.792,-80.056,-176.273,9.012,148.732
C08840=1160.676,361.039,-80.090,-176.270,9.016,148.732
C08841=1160.672,361.287,-80.124,-176.268,9.020,148.733
C08842=1160.668,361.534,-80.159,-176.266,9.024,148.733
C08843=1160.664,361.782,-80.194,-176.264,9.028,148.733
C08844=1160.660,362.029,-80.229,-176.261,9.032,148.734
C08845=1160.656,362.277,-80.264,-176.259,9.035,148.734
C08846=1160.653,362.524,-80.299,-176.256,9.039,148.734
C08847=1160.648,362.771,-80.334,-176.254,9.043,148.735
C08848=1160.644,363.019,-80.369,-176.251,9.047,148.735
C08849=1160.640,363.267,-80.403,-176.249,9.050,148.735
C08850=1160.636,363.514,-80.439,-176.247,9.055,148.736
C08851=1160.633,363.762,-80.473,-176.244,9.058,148.736
C08852=1160.629,364.009,-80.508,-176.242,9.062,148.736
C08853=1160.625,364.257,-80.543,-176.240,9.066,148.737
C08854=1160.621,364.504,-80.578,-176.237,9.070,148.737
C08855=1160.617,364.752,-80.613,-176.235,9.073,148.737
C08856=1160.613,364.999,-80.648,-176.232,9.078,148.738
C08857=1160.609,365.282,-80.688,-176.230,9.082,148.738
C08858=1160.604,365.564,-80.729,-176.227,9.086,148.739
C08859=1160.599,365.847,-80.768,-176.225,9.091,148.739
C08860=1160.595,366.129,-80.808,-176.222,9.095,148.740
C08861=1160.591,366.377,-80.843,-176.220,9.100,148.740
C08862=1160.587,366.625,-80.879,-176.217,9.103,148.740
C08863=1160.583,366.872,-80.914,-176.215,9.107,148.741
C08864=1160.579,367.120,-80.949,-176.213,9.111,148.741
C08865=1160.575,367.367,-80.984,-176.210,9.115,148.741
C08866=1160.572,367.615,-81.020,-176.208,9.119,148.742
C08867=1160.567,367.862,-81.054,-176.206,9.123,148.742
C08868=1160.564,368.110,-81.090,-176.204,9.127,148.743
C08869=1160.560,368.357,-81.125,-176.201,9.131,148.743
C08870=1160.555,368.604,-81.160,-176.200,9.135,148.744
C08871=1160.552,368.852,-81.195,-176.197,9.138,148.744
C08872=1160.548,369.099,-81.231,-176.195,9.142,148.744
C08873=1160.544,369.347,-81.266,-176.193,9.146,148.745
C08874=1160.539,369.594,-81.302,-176.191,9.150,148.745
C08875=1160.535,369.842,-81.337,-176.189,9.154,148.746
C08876=1160.532,370.090,-81.373,-176.186,9.158,148.746
C08877=1160.527,370.337,-81.408,-176.184,9.162,148.747
C08878=1160.524,370.584,-81.443,-176.182,9.166,148.747
C08879=1160.520,370.832,-81.479,-176.180,9.170,148.748
C08880=1160.516,371.079,-81.514,-176.179,9.174,148.748
C08881=1160.513,371.327,-81.549,-176.177,9.177,148.748
C08882=1160.508,371.574,-81.584,-176.174,9.182,148.749
C08883=1160.505,371.821,-81.620,-176.172,9.185,148.749
C08884=1160.500,372.069,-81.656,-176.171,9.189,148.750
C08885=1160.497,372.317,-81.692,-176.168,9.194,148.750
C08886=1160.492,372.564,-81.727,-176.167,9.197,148.751
C08887=1160.489,372.811,-81.762,-176.165,9.201,148.751
C08888=1160.485,373.059,-81.798,-176.163,9.205,148.752
C08889=1160.481,373.306,-81.833,-176.161,9.209,148.752
C08890=1160.477,373.554,-81.870,-176.159,9.213,148.753
C08891=1160.473,373.801,-81.905,-176.158,9.217,148.753
C08892=1160.469,374.048,-81.940,-176.156,9.221,148.754
C08893=1160.465,374.296,-81.976,-176.154,9.224,148.755
C08894=1160.462,374.543,-82.011,-176.153,9.228,148.755
C08895=1160.457,374.791,-82.048,-176.150,9.233,148.756
C08896=1160.454,375.038,-82.083,-176.149,9.236,148.756
C08897=1160.450,375.286,-82.119,-176.147,9.240,148.757
C08898=1160.446,375.532,-82.155,-176.146,9.244,148.757
C08899=1160.442,375.780,-82.191,-176.144,9.248,148.758
C08900=1160.438,376.027,-82.226,-176.143,9.252,148.759
C08901=1160.434,376.275,-82.262,-176.141,9.256,148.759
C08902=1160.431,376.522,-82.297,-176.139,9.259,148.760
C08903=1160.426,376.770,-82.334,-176.138,9.263,148.760
C08904=1160.423,377.017,-82.370,-176.136,9.267,148.761
C08905=1160.419,377.264,-82.405,-176.135,9.271,148.761
C08906=1160.414,377.512,-82.441,-176.134,9.275,148.762
C08907=1160.410,377.759,-82.477,-176.132,9.279,148.763
C08908=1160.407,378.007,-82.512,-176.131,9.283,148.763
C08909=1160.403,378.254,-82.549,-176.129,9.287,148.764
C08910=1160.399,378.501,-82.585,-176.128,9.290,148.765
C08911=1160.395,378.749,-82.620,-176.127,9.294,148.765
C08912=1160.391,378.997,-82.656,-176.126,9.298,148.766
C08913=1160.388,379.244,-82.693,-176.124,9.302,148.767
C08914=1160.383,379.490,-82.728,-176.123,9.306,148.767
C08915=1160.379,379.738,-82.764,-176.123,9.309,148.768
C08916=1160.376,379.985,-82.800,-176.121,9.313,148.769
C08917=1160.371,380.233,-82.836,-176.120,9.317,148.769
C08918=1160.368,380.480,-82.872,-176.119,9.320,148.770
C08919=1160.364,380.727,-82.908,-176.118,9.324,148.771
C08920=1160.360,380.975,-82.944,-176.117,9.328,148.771
C08921=1160.356,381.223,-82.980,-176.116,9.331,148.772
C08922=1160.352,381.470,-83.017,-176.115,9.336,148.773
C08923=1160.348,381.717,-83.052,-176.114,9.339,148.773
C08924=1160.345,381.965,-83.088,-176.113,9.343,148.774
C08925=1160.341,382.212,-83.125,-176.113,9.346,148.775
C08926=1160.337,382.460,-83.160,-176.112,9.349,148.776
C08927=1160.333,382.707,-83.197,-176.111,9.353,148.776
C08928=1160.329,382.954,-83.233,-176.110,9.357,148.777
C08929=1160.325,383.202,-83.269,-176.110,9.360,148.778
C08930=1160.321,383.449,-83.305,-176.108,9.364,148.779
C08931=1160.317,383.697,-83.341,-176.108,9.368,148.779
C08932=1160.314,383.944,-83.377,-176.107,9.371,148.780
C08933=1160.309,384.191,-83.414,-176.107,9.374,148.781
C08934=1160.306,384.438,-83.450,-176.107,9.378,148.782
C08935=1160.302,384.686,-83.486,-176.106,9.382,148.782
C08936=1160.298,384.933,-83.522,-176.105,9.385,148.783
C08937=1160.294,385.181,-83.558,-176.105,9.389,148.784
C08938=1160.290,385.427,-83.594,-176.104,9.392,148.785
C08939=1160.285,385.675,-83.630,-176.104,9.395,148.785
C08940=1160.282,385.922,-83.667,-176.104,9.398,148.786
C08941=1160.278,386.170,-83.703,-176.103,9.401,148.787
C08942=1160.275,386.417,-83.739,-176.103,9.405,148.788
C08943=1160.271,386.665,-83.776,-176.103,9.409,148.789
C08944=1160.267,386.912,-83.812,-176.103,9.412,148.789
C08945=1160.263,387.159,-83.849,-176.103,9.414,148.790
C08946=1160.259,387.406,-83.884,-176.103,9.418,148.791
C08947=1160.255,387.654,-83.921,-176.103,9.421,148.792
C08948=1160.252,387.901,-83.957,-176.102,9.424,148.793
C08949=1160.248,388.148,-83.993,-176.102,9.428,148.794
C08950=1160.244,388.396,-84.029,-176.102,9.430,148.794
C08951=1160.240,388.643,-84.066,-176.102,9.434,148.795
C08952=1160.236,388.890,-84.102,-176.103,9.437,148.796
C08953=1160.232,389.138,-84.138,-176.103,9.439,148.797
C08954=1160.229,389.385,-84.175,-176.102,9.443,148.797
C08955=1160.224,389.632,-84.211,-176.103,9.445,148.798
C08956=1160.220,389.880,-84.248,-176.103,9.448,148.799
C08957=1160.217,390.126,-84.284,-176.103,9.452,148.800
C08958=1160.212,390.374,-84.320,-176.103,9.454,148.801
C08959=1160.209,390.621,-84.356,-176.104,9.457,148.802
C08960=1160.205,390.868,-84.393,-176.104,9.460,148.802
C08961=1160.201,391.154,-84.434,-176.104,9.463,148.803
C08962=1160.196,391.440,-84.476,-176.104,9.466,148.804
C08963=1160.192,391.725,-84.519,-176.105,9.469,148.805
C08964=1160.187,392.011,-84.561,-176.105,9.473,148.806
C08965=1160.183,392.258,-84.597,-176.105,9.476,148.807
C08966=1160.179,392.505,-84.634,-176.105,9.478,148.808
C08967=1160.175,392.753,-84.670,-176.106,9.481,148.809
C08968=1160.172,393.001,-84.706,-176.107,9.483,148.809
C08969=1160.168,393.248,-84.743,-176.107,9.486,148.810
C08970=1160.164,393.495,-84.779,-176.108,9.489,148.811
C08971=1160.160,393.743,-84.816,-176.108,9.491,148.812
C08972=1160.157,393.990,-84.852,-176.109,9.494,148.813
C08973=1160.153,394.237,-84.888,-176.109,9.497,148.813
C08974=1160.148,394.485,-84.925,-176.110,9.499,148.814
C08975=1160.145,394.731,-84.961,-176.110,9.501,148.815
C08976=1160.141,394.979,-84.997,-176.110,9.504,148.816
C08977=1160.137,395.226,-85.034,-176.111,9.507,148.817
C08978=1160.133,395.473,-85.071,-176.112,9.509,148.817
C08979=1160.129,395.720,-85.107,-176.112,9.511,148.818
C08980=1160.125,395.968,-85.143,-176.113,9.513,148.819
C08981=1160.121,396.215,-85.180,-176.113,9.516,148.820
C08982=1160.117,396.462,-85.217,-176.114,9.519,148.821
C08983=1160.114,396.710,-85.252,-176.114,9.521,148.821
C08984=1160.110,396.957,-85.289,-176.115,9.523,148.822
C08985=1160.106,397.205,-85.326,-176.116,9.525,148.823
C08986=1160.103,397.452,-85.363,-176.116,9.528,148.824
C08987=1160.098,397.700,-85.399,-176.117,9.530,148.824
C08988=1160.094,397.947,-85.436,-176.117,9.533,148.825
C08989=1160.091,398.194,-85.472,-176.118,9.534,148.826
C08990=1160.087,398.441,-85.509,-176.119,9.537,148.827
C08991=1160.083,398.688,-85.544,-176.119,9.539,148.827
C08992=1160.079,398.936,-85.581,-176.120,9.542,148.828
C08993=1160.075,399.183,-85.618,-176.121,9.544,148.829
C08994=1160.071,399.430,-85.653,-176.121,9.545,148.830
C08995=1160.067,399.677,-85.690,-176.122,9.548,148.830
C08996=1160.063,399.925,-85.727,-176.123,9.550,148.831
C08997=1160.060,400.172,-85.763,-176.123,9.552,148.832
C08998=1160.055,400.419,-85.800,-176.124,9.555,148.833
C08999=1160.052,400.667,-85.837,-176.125,9.556,148.833
C09000=1160.048,400.914,-85.873,-176.125,9.558,148.834
C09001=1160.044,401.161,-85.910,-176.126,9.561,148.835
C09002=1160.040,401.409,-85.946,-176.127,9.563,148.836
C09003=1160.037,401.656,-85.982,-176.127,9.565,148.836
C09004=1160.032,401.903,-86.019,-176.128,9.567,148.837
C09005=1160.028,402.150,-86.056,-176.128,9.569,148.838
C09006=1160.025,402.397,-86.092,-176.129,9.571,148.838
C09007=1160.021,402.645,-86.128,-176.130,9.573,148.839
C09008=1160.017,402.892,-86.165,-176.131,9.575,148.840
C09009=1160.013,403.139,-86.202,-176.131,9.577,148.841
C09010=1160.009,403.386,-86.238,-176.132,9.579,148.841
C09011=1160.005,403.635,-86.275,-176.133,9.581,148.842
C09012=1160.002,403.882,-86.311,-176.134,9.583,148.843
C09013=1159.998,404.129,-86.348,-176.134,9.585,148.843
C09014=1159.994,404.376,-86.385,-176.134,9.587,148.844
C09015=1159.990,404.624,-86.420,-176.135,9.589,148.845
C09016=1159.986,404.871,-86.457,-176.136,9.591,148.845
C09017=1159.982,405.118,-86.494,-176.137,9.593,148.846
C09018=1159.979,405.365,-86.530,-176.138,9.595,148.847
C09019=1159.974,405.612,-86.567,-176.138,9.596,148.848
C09020=1159.970,405.860,-86.603,-176.138,9.599,148.848
C09021=1159.967,406.107,-86.640,-176.139,9.601,148.849
C09022=1159.963,406.355,-86.677,-176.140,9.602,148.850
C09023=1159.959,406.602,-86.714,-176.141,9.604,148.850
C09024=1159.956,406.849,-86.750,-176.141,9.606,148.851
C09025=1159.951,407.097,-86.786,-176.142,9.608,148.851
C09026=1159.947,407.344,-86.823,-176.143,9.609,148.852
C09027=1159.944,407.591,-86.859,-176.143,9.611,148.853
C09028=1159.940,407.838,-86.896,-176.143,9.614,148.853
C09029=1159.936,408.085,-86.933,-176.144,9.615,148.854
C09030=1159.932,408.332,-86.969,-176.145,9.617,148.855
C09031=1159.928,408.580,-87.005,-176.146,9.619,148.855
C09032=1159.924,408.828,-87.043,-176.146,9.621,148.856
C09033=1159.921,409.074,-87.079,-176.147,9.622,148.857
C09034=1159.917,409.322,-87.116,-176.148,9.624,148.857
C09035=1159.913,409.569,-87.152,-176.148,9.626,148.858
C09036=1159.909,409.816,-87.188,-176.148,9.628,148.859
C09037=1159.905,410.064,-87.225,-176.149,9.630,148.859
C09038=1159.901,410.311,-87.262,-176.150,9.632,148.860
C09039=1159.898,410.558,-87.298,-176.151,9.634,148.861
C09040=1159.893,410.805,-87.334,-176.151,9.635,148.861
C09041=1159.889,411.053,-87.371,-176.152,9.637,148.862
C09042=1159.886,411.300,-87.408,-176.152,9.639,148.862
C09043=1159.882,411.547,-87.445,-176.153,9.640,148.863
C09044=1159.878,411.795,-87.482,-176.154,9.642,148.864
C09045=1159.874,412.042,-87.518,-176.154,9.645,148.864
C09046=1159.870,412.289,-87.554,-176.154,9.646,148.865
C09047=1159.866,412.536,-87.591,-176.155,9.648,148.865
C09048=1159.862,412.784,-87.628,-176.155,9.650,148.866
C09049=1159.859,413.030,-87.664,-176.156,9.651,148.867
C09050=1159.855,413.278,-87.701,-176.157,9.653,148.867
C09051=1159.850,413.526,-87.737,-176.157,9.655,148.868
C09052=1159.848,413.773,-87.774,-176.158,9.656,148.868
C09053=1159.844,414.020,-87.810,-176.158,9.659,148.869
C09054=1159.839,414.267,-87.847,-176.159,9.661,148.870
C09055=1159.835,414.515,-87.884,-176.159,9.662,148.870
C09056=1159.832,414.762,-87.920,-176.160,9.664,148.871
C09057=1159.828,415.009,-87.957,-176.160,9.666,148.872
C09058=1159.825,415.257,-87.993,-176.161,9.667,148.872
C09059=1159.822,415.504,-88.029,-176.161,9.669,148.873
C09060=1159.820,415.751,-88.067,-176.161,9.671,148.873
C09061=1159.819,416.117,-88.120,-176.162,9.673,148.874
C09062=1159.820,416.483,-88.173,-176.162,9.676,148.875
C09063=1159.823,416.848,-88.227,-176.164,9.678,148.876
C09064=1159.828,417.213,-88.279,-176.164,9.681,148.876
C09065=1159.407,417.215,-88.326,-176.167,9.692,148.880
C09066=1159.402,416.847,-88.273,-176.166,9.689,148.879
C09067=1159.399,416.478,-88.220,-176.166,9.687,148.879
C09068=1159.398,416.109,-88.165,-176.165,9.684,148.878
C09069=1159.400,415.739,-88.111,-176.164,9.682,148.877
C09070=1159.401,415.493,-88.075,-176.164,9.681,148.876
C09071=1159.403,415.246,-88.039,-176.164,9.678,148.876
C09072=1159.407,414.998,-88.001,-176.163,9.676,148.875
C09073=1159.411,414.750,-87.965,-176.163,9.675,148.875
C09074=1159.415,414.503,-87.929,-176.162,9.673,148.874
C09075=1159.419,414.256,-87.892,-176.161,9.671,148.873
C09076=1159.423,414.009,-87.855,-176.161,9.670,148.873
C09077=1159.426,413.762,-87.819,-176.160,9.668,148.872
C09078=1159.430,413.514,-87.782,-176.160,9.666,148.872
C09079=1159.434,413.267,-87.745,-176.160,9.664,148.871
C09080=1159.438,413.019,-87.708,-176.159,9.662,148.870
C09081=1159.442,412.772,-87.672,-176.158,9.660,148.870
C09082=1159.446,412.525,-87.636,-176.158,9.659,148.869
C09083=1159.450,412.278,-87.599,-176.157,9.657,148.869
C09084=1159.453,412.031,-87.563,-176.156,9.655,148.868
C09085=1159.457,411.783,-87.526,-176.156,9.654,148.867
C09086=1159.461,411.536,-87.489,-176.156,9.651,148.867
C09087=1159.465,411.289,-87.453,-176.155,9.649,148.866
C09088=1159.469,411.042,-87.416,-176.155,9.648,148.865
C09089=1159.472,410.794,-87.379,-176.154,9.646,148.865
C09090=1159.477,410.546,-87.342,-176.153,9.644,148.864
C09091=1159.480,410.300,-87.306,-176.153,9.643,148.864
C09092=1159.484,410.052,-87.270,-176.152,9.641,148.863
C09093=1159.488,409.805,-87.233,-176.151,9.639,148.862
C09094=1159.492,409.558,-87.197,-176.151,9.637,148.862
C09095=1159.496,409.311,-87.160,-176.150,9.636,148.861
C09096=1159.500,409.063,-87.123,-176.150,9.633,148.860
C09097=1159.503,408.816,-87.087,-176.149,9.631,148.860
C09098=1159.508,408.569,-87.051,-176.148,9.630,148.859
C09099=1159.511,408.321,-87.013,-176.148,9.628,148.858
C09100=1159.515,408.074,-86.977,-176.147,9.626,148.858
C09101=1159.519,407.827,-86.940,-176.146,9.624,148.857
C09102=1159.523,407.579,-86.903,-176.146,9.623,148.856
C09103=1159.526,407.332,-86.868,-176.145,9.621,148.856
C09104=1159.531,407.085,-86.831,-176.144,9.619,148.855
C09105=1159.535,406.838,-86.794,-176.144,9.616,148.854
C09106=1159.539,406.590,-86.757,-176.143,9.615,148.854
C09107=1159.542,406.344,-86.721,-176.143,9.613,148.853
C09108=1159.546,406.096,-86.685,-176.142,9.611,148.852
C09109=1159.550,405.848,-86.648,-176.141,9.610,148.852
C09110=1159.553,405.601,-86.611,-176.141,9.608,148.851
C09111=1159.557,405.354,-86.575,-176.139,9.606,148.850
C09112=1159.562,405.107,-86.538,-176.139,9.603,148.850
C09113=1159.565,404.859,-86.502,-176.139,9.601,148.849
C09114=1159.569,404.612,-86.465,-176.138,9.600,148.848
C09115=1159.573,404.365,-86.428,-176.137,9.598,148.848
C09116=1159.577,404.118,-86.392,-176.137,9.596,148.847
C09117=1159.581,403.871,-86.355,-176.135,9.594,148.846
C09118=1159.585,403.623,-86.319,-176.135,9.592,148.845
C09119=1159.588,403.375,-86.283,-176.135,9.590,148.845
C09120=1159.592,403.128,-86.246,-176.134,9.588,148.844
C09121=1159.596,402.881,-86.209,-176.133,9.586,148.843
C09122=1159.600,402.633,-86.173,-176.132,9.584,148.843
C09123=1159.604,402.386,-86.136,-176.132,9.582,148.842
C09124=1159.608,402.139,-86.100,-176.131,9.580,148.841
C09125=1159.611,401.892,-86.063,-176.130,9.578,148.840
C09126=1159.615,401.645,-86.026,-176.129,9.576,148.840
C09127=1159.620,401.397,-85.990,-176.129,9.574,148.839
C09128=1159.623,401.150,-85.954,-176.128,9.571,148.838
C09129=1159.627,400.903,-85.917,-176.127,9.570,148.838
C09130=1159.631,400.656,-85.880,-176.127,9.568,148.837
C09131=1159.634,400.408,-85.844,-176.126,9.565,148.836
C09132=1159.639,400.160,-85.808,-176.125,9.563,148.835
C09133=1159.643,399.913,-85.771,-176.124,9.561,148.835
C09134=1159.646,399.666,-85.734,-176.124,9.559,148.834
C09135=1159.650,399.419,-85.698,-176.124,9.557,148.833
C09136=1159.655,399.171,-85.661,-176.122,9.555,148.832
C09137=1159.658,398.924,-85.625,-176.122,9.552,148.832
C09138=1159.662,398.677,-85.588,-176.121,9.550,148.831
C09139=1159.666,398.430,-85.553,-176.121,9.548,148.830
C09140=1159.670,398.183,-85.516,-176.120,9.546,148.829
C09141=1159.674,397.935,-85.479,-176.119,9.544,148.829
C09142=1159.677,397.689,-85.443,-176.119,9.541,148.828
C09143=1159.681,397.440,-85.406,-176.118,9.539,148.827
C09144=1159.685,397.193,-85.369,-176.117,9.536,148.826
C09145=1159.688,396.946,-85.333,-176.117,9.535,148.826
C09146=1159.693,396.699,-85.296,-176.116,9.532,148.825
C09147=1159.697,396.451,-85.260,-176.115,9.530,148.824
